	(* Switch S27 *)
	nAX5203DigitalInputs.3;
	

(* Axis 1-4 aktiv *)
	bLedH16 := ((Axis1.fbAxis.bMoveAbsBusy
					OR Axis2.fbAxis.bMoveAbsBusy
						OR Axis3.fbAxis.bMoveAbsBusy
							OR Axis4.fbAxis.bMoveAbsBusy)
				AND bClock500ms)
				OR (Axis1.fbAxis.bMoveAbsDone
					AND Axis2.fbAxis.bMoveAbsDone
						AND Axis3.fbAxis.bMoveAbsDone
							AND Axis4.fbAxis.bMoveAbsDone);

(* Axis 1-4 coupled *)
	bLedH17 := ((stAxis1.Status.Coupled
					OR stAxis2.Status.Coupled
						OR stAxis3.Status.Coupled
							OR stAxis4.Status.Coupled)
				AND bClock500ms)
				OR bSwitchS17;
				
(* Axis 1-4 reversing sequence busy *)		
	bLedH20 := (Axis1.fbAxis.bRevSeqBusy
					OR Axis2.fbAxis.bRevSeqBusy
						OR Axis3.fbAxis.bRevSeqBusy
							OR Axis4.fbAxis.bRevSeqBusy)
				AND bClock500ms;

(* Axis 1-4 error detectet *)
	bLedH21 := (stAxis1.Status.Error
					OR stAxis2.Status.Error
						OR stAxis3.Status.Error
							OR stAxis4.Status.Error)
				AND bClock500ms;

(* End *)

END_PROGRAM

// ---- POUs/Motion/Axis1.TcPOU
PROGRAM Axis1
VAR

	sAxisDescription						:STRING	:= 'Axis 1 - EL7037 - AS1020-0120';	

(* Axis - basic functions *)
	fbAxis									:FB_Axis;
	fMoveAbsPosition						:LREAL;				(* Target position *)
	fMoveAbsVelocity						:LREAL	:= 500.0;	(* Target speed axis 1 max. 3600.0 Degree/s *)
	bStartMoveAbs							:BOOL;
	bMoveAbsBusy							:BOOL;
	bMoveAbsDone							:BOOL;
	bAxisErr								:BOOL;
	nAxisErrId								:DWORD;
	bReset									:BOOL;
	bStop									:BOOL;
	bStopAxisDone							:BOOL;
	bStopAxisBusy							:BOOL;
	bRevSeqStart							:BOOL;
	bStartparameterSet						:BOOL;
	
(* Test - change target position *)
	bTestChangeTargetPos					:BOOL;				(* Test - change target position *)
	bMaxPositionReached						:BOOL;
	
(* Homing *)
	fbHomingAxis							:MC_Home;
	fHomingPosition							:LREAL	:= 331.00;

(* Touch Probe *)
	fbTouchProbe							:MC_TouchProbe;
	stTriggerInput							:TRIGGER_REF;
	bTouchProbeDone							:BOOL;
	bTouchProbeBusy							:BOOL;
	bTouchProbeComAb						:BOOL;
	bTouchProbeErr							:BOOL;
	bTouchProbeErrId						:UDINT;
	fRecordedPosition 						:LREAL;
	stRecordedData							:MC_TouchProbeRecordedData;	

(* Couple Axis on Handwheel *)
	fbGearIn								:MC_GearIn;
	bGearInDone								:BOOL;
	bAxisCoupled							:BOOL;

(* Uncouple Axis *)
	fbGearOut								:MC_GearOut;
	bGearOutDone							:BOOL;

END_VAR
(* End *)

(* Axis 1 *)

(* Axis - basic functions  *)

	IF NOT bStartparameterSet
	THEN
		(* Startup Parameter reversing sequence *)
		fbAxis.fRevSeqTargetPos1	:= 720.0;
		fbAxis.fRevSeqTargetVelo1	:= 500.0;
		fbAxis.fRevSeqTargetPos2	:= 0.0;
		fbAxis.fRevSeqTargetVelo2	:= 3000.0;
		fbAxis.nRevSeqIdleTime		:= 500;
		bStartparameterSet			:= TRUE;
	END_IF
		
	fbAxis(
		bPowerEnable		:= 	bSwitchS12,
		fPowerOverride		:= 	F_Scaling(nAnalogInR10, 100.0, 32767.0),
		bMoveAbsExecute		:= 	(bStartMoveAbs OR bSwitchS16) AND NOT stAxis1.Status.Coupled,
		fMoveAbsPosition	:= 	fMoveAbsPosition,
		fMoveAbsVelocity	:= 	fMoveAbsVelocity,
		bReset				:= 	bReset OR bSwitchS21,
		bStopAxis			:= 	bStop,
		bRevSeqStart		:=  (bSwitchS20 OR bRevSeqStart) AND fbAxis.bPowerStatus, 
		stAxis				:= 	stAxis1,
		bPowerStatus		=> 	bLedH12,
		bMoveAbsDone		=> 	bMoveAbsDone,
		bMoveAbsBusy		=> 	bMoveAbsBusy,
		bAxisErr			=> 	bAxisErr,
		nAxisErrId			=> 	nAxisErrId,
		bStopAxisDone		=> 	bStopAxisDone,
		bStopAxisBusy		=> 	bStopAxisBusy);
		

(* Test - change target position - Axis *)
	IF bTestChangeTargetPos
		AND (fMoveAbsPosition <= stAxis1.NcToPlc.ActPos)
			AND NOT bMaxPositionReached
	THEN
		fMoveAbsPosition := fMoveAbsPosition + 180.0;
	ELSE
		IF bTestChangeTargetPos
			AND (fMoveAbsPosition >= 3600.0)
		THEN
			fMoveAbsPosition 	:= 0.0;
			bMaxPositionReached	:= TRUE;
		END_IF
	END_IF

	IF bTestChangeTargetPos
		AND (stAxis1.NcToPlc.ActPos < 1.0)
	THEN
		bMaxPositionReached	:= FALSE;
	END_IF

	IF bSwitchS17
	THEN
		bMaxPositionReached	:= FALSE;
		fMoveAbsPosition 	:= 0.0;
	END_IF
	
(* Homing Axis *)
	fbHomingAxis(
		Execute			:= 	bSwitchS23 AND fbAxis.bPowerStatus,
		Position		:= 	fHomingPosition,
		HomingMode		:= 	MC_DefaultHoming,
		BufferMode		:= 	,
		Options			:= 	,
		bCalibrationCam	:= 	bStepperReferenceCam,
		Axis			:= 	stAxis1,
		Done			=> 	,
		Busy			=> 	,
		Active			=> 	,
		CommandAborted	=> 	,
		Error			=> 	,
		ErrorID			=> 	);
		
		
	bLedH23 :=	(bClock1s 
					AND NOT stAxis1.Status.Homed
					AND fbAxis.bPowerStatus
					AND NOT fbHomingAxis.Busy)
				OR (bClock500ms 
					AND fbHomingAxis.Busy)
				OR fbHomingAxis.Done;
					

(* Touch Probe *)
	stTriggerInput.EncoderID 		:= 1;
	stTriggerInput.TouchProbe 		:= TouchProbe1;
	stTriggerInput.SignalSource 	:= SignalSource_Default;
	stTriggerInput.Edge 			:= RisingEdge;
	stTriggerInput.Mode 			:= TOUCHPROBEMODE_SINGLE;
	stTriggerInput.ModuloPositions 	:= FALSE;

	fbTouchProbe(
		Execute			:= 	bSwitchS24,
		WindowOnly		:= 	,
		FirstPosition	:= 	,
		LastPosition	:= 	,
		Axis			:= 	stAxis1,
		TriggerInput	:= 	stTriggerInput,
		Done			=> 	bTouchProbeDone,
		Busy			=> 	bTouchProbeBusy,
		CommandAborted	=> 	bTouchProbeComAb,
		Error			=> 	bTouchProbeErr,
		ErrorID			=> 	bTouchProbeErrId,
		RecordedPosition=> 	fRecordedPosition,
		RecordedData	=>	stRecordedData);
	
	bLedH24 :=	(bClock500ms 
					AND fbTouchProbe.Busy)
						OR fbTouchProbe.Done;

(* Couple Axis on Handwheel *)
	fbGearIn(
		Execute			:= 	bHandwheelSwitchS28,
		RatioNumerator	:= 	1,
		RatioDenominator:= 	1,
		Acceleration	:= 	,
		Deceleration	:= 	,
		Jerk			:= 	,
		BufferMode		:= 	,
		Options			:= 	,
		Master			:= 	stAxis5,
		Slave			:= 	stAxis1,
		InGear			=> 	bGearInDone,
		Busy			=> 	,
		Active			=> 	,
		CommandAborted	=> 	,
		Error			=> 	,
		ErrorID			=> 	);

(* Axis coupled *)
	bAxisCoupled := stAxis1.Status.Coupled;

(* Uncouple Axis *)
	fbGearOut(
		Execute	:= 	bSwitchS17,
		Options	:= 	,
		Slave	:= 	stAxis1,
		Done	=> 	bGearOutDone,
		Busy	=> 	,
		Error	=> 	,
		ErrorID	=> 	);
	
(* End *)

END_PROGRAM

// ---- POUs/Motion/Components/FB_Axis.TcPOU
FUNCTION_BLOCK FB_Axis
VAR_INPUT
	
	bPowerEnable							:BOOL;
	fPowerOverride							:LREAL;
	bMoveAbsExecute							:BOOL;
	fMoveAbsPosition						:LREAL;
	fMoveAbsVelocity						:LREAL;
	bReset									:BOOL;
	bStopAxis								:BOOL;
	bRevSeqStart							:BOOL;
	bRevSeqStop								:BOOL;
	fRevSeqTargetPos1						:LREAL; 
	fRevSeqTargetVelo1						:LREAL;	 
	fRevSeqTargetPos2						:LREAL;	 
	fRevSeqTargetVelo2						:LREAL; 
	nRevSeqIdleTime							:UINT;
	
END_VAR
VAR_OUTPUT

	bPowerStatus							:BOOL;
	bMoveAbsDone							:BOOL;
	bMoveAbsBusy							:BOOL;
	bAxisErr								:BOOL;
	nAxisErrId								:DWORD;
	bStopAxisDone							:BOOL;
	bStopAxisBusy							:BOOL;
	bRevSeqDone								:BOOL;
	bRevSeqBusy								:BOOL;
	
END_VAR
VAR_IN_OUT

	stAxis									:Axis_Ref;

END_VAR
VAR

	fbMcPower								:MC_Power;
	fbMoveAbsolute							:MC_MoveAbsolute;
	fbReadAxisError							:MC_ReadAxisError;
	fbReset									:MC_Reset;
	fbStop									:MC_Stop;
	fbReversingSequence						:FB_ReversingSequence;

END_VAR
(* End *)

(* FB_Axis *)

(* Read status of the axis *)
	stAxis.ReadStatus();

(* Enable axis *)
	fbMcPower(
		Enable			:= 	bPowerEnable,
		Enable_Positive	:= 	bPowerEnable,
		Enable_Negative	:= 	bPowerEnable,
		Override		:= 	fPowerOverride,
		Axis			:= 	stAxis,
		Status			=> 	bPowerStatus);

(* Start axis at an absolute position *)
	fbMoveAbsolute(
		Execute		:=	bMoveAbsExecute,
		Position	:=	fMoveAbsPosition,
		Velocity	:=	fMoveAbsVelocity,
		Axis		:=	stAxis,
		Done		=>	bMoveAbsDone,
		Busy		=>	bMoveAbsBusy);

(* Read the error code of the axis *)
	fbReadAxisError(
		Enable		:=	TRUE,
		Axis		:=	stAxis,
		AxisErrorID	=>	nAxisErrId);
		
	bAxisErr := nAxisErrId <> 0;

(* Reset axis in case of failure *)
	fbReset(
		Execute		:= 	bReset,
		Axis		:= 	stAxis);

(* Stop axis *)
	fbStop(
		Execute 	:=	bStopAxis,
		Axis		:=	stAxis,
		Done		=>	bStopAxisDone,
		Busy		=>	bStopAxisBusy);

(* Axis reversing sequence *)	
	fbReversingSequence(
		bStart				:= 	bRevSeqStart,
		bStop				:= 	bRevSeqStop,
		fTargetPosition1	:= 	fRevSeqTargetPos1,
		fTargetVelocity1	:= 	fRevSeqTargetVelo1,
		fTargetPosition2	:= 	fRevSeqTargetPos2,
		fTargetVelocity2	:= 	fRevSeqTargetVelo2,
		tIdleTime			:= 	TO_TIME(nRevSeqIdleTime),
		bDone				=> 	bRevSeqDone,
		bBusy				=> 	bRevSeqBusy,
		bErr				=> 	,
		nErrID				=> 	,
		stAxis				:= 	stAxis);
		
(* End *)

END_FUNCTION_BLOCK

// ---- POUs/Motion/Components/FB_ReversingSequence.TcPOU
FUNCTION_BLOCK FB_ReversingSequence
VAR_INPUT
	
	bStart									:BOOL;
	bStop									:BOOL;	
	fTargetPosition1						:LREAL;
	fTargetVelocity1						:LREAL;
	fTargetPosition2						:LREAL;
	fTargetVelocity2						:LREAL;
	tIdleTime								:TIME;
	
END_VAR
VAR_OUTPUT
	
	bDone									:BOOL;
	bBusy									:BOOL;
	bErr									:BOOL;
	nErrID									:UDINT;
	
END_VAR
VAR_IN_OUT

	stAxis									:Axis_Ref;

END_VAR
VAR
	
	eStateRevSeq							:E_AxisReversingSequence;
	eRevSeqErrStep							:E_AxisReversingSequence := eAxisRevSeq_NoError;
	fbTimerIdleTime							:TON;
	fbMoveAbsolute							:MC_MoveAbsolute;
	fbStop									:MC_Stop;

END_VAR
(* End *)

(* Reversing sequence axis *)

	CASE eStateRevSeq OF

		eAxisRevSeq_Start			:	(* Wait for start *)
		
			bDone := FALSE;
			bBusy := FALSE;
			
			IF bStart
			THEN

				bBusy 		 := TRUE;
				eStateRevSeq := eAxisRevSeq_Init;
				
			END_IF		


		eAxisRevSeq_Init			:	(* Initialize *)
		
			fbMoveAbsolute(
				Axis	 := stAxis, 
				Execute	 := FALSE);
				
			fbTimerIdleTime(
				IN	 	 :=	FALSE);
			
			fbStop(
				Axis	 :=	stAxis,
				Execute	 :=	FALSE);
				
			eStateRevSeq := eAxisRevSeq_AxisStartPos1;


		eAxisRevSeq_AxisStartPos1	:	(* Start axis to position 1 *)
		
			fbMoveAbsolute(
				Axis		:= stAxis, 
				Execute		:= TRUE, 
				Position	:= fTargetPosition1, 
				Velocity	:= fTargetVelocity1, 
				ErrorID		=> nErrID);
			
		
			IF NOT fbMoveAbsolute.Busy
				AND NOT fbMoveAbsolute.Error
			THEN
			
				fbMoveAbsolute(
					Axis		:= stAxis, 
					Execute		:= FALSE);
				eStateRevSeq := eAxisRevSeq_IdleTime1;

			ELSIF bStop
			THEN

				fbMoveAbsolute(
					Axis	 := stAxis, 
					Execute	 := FALSE);
				eStateRevSeq := eAxisRevSeq_AxisStop;

			ELSIF NOT fbMoveAbsolute.Busy
					AND fbMoveAbsolute.Error
			THEN

				eRevSeqErrStep := eStateRevSeq;
				eStateRevSeq   := eAxisRevSeq_ErrorStep;

			END_IF


		eAxisRevSeq_IdleTime1		:	(* delayed restart *)
		
			fbTimerIdleTime(
				IN	:=	TRUE, 
				PT	:= 	tIdleTime);

			IF NOT bStop			
				AND fbTimerIdleTime.Q 
			THEN

				fbTimerIdleTime(IN	:=	FALSE);
				eStateRevSeq := eAxisRevSeq_AxisStartPos2;

			ELSIF bStop
			THEN

				eStateRevSeq := eAxisRevSeq_Done;

			END_IF


		eAxisRevSeq_AxisStartPos2	:	(* Start axis to position 2 *)
		
			fbMoveAbsolute(
				Axis		:= stAxis, 
				Execute		:= TRUE, 
				Position	:= fTargetPosition2, 
				Velocity	:= fTargetVelocity2, 
				ErrorID		=> nErrID);
			
		
			IF NOT fbMoveAbsolute.Busy
				AND NOT fbMoveAbsolute.Error
			THEN
				fbMoveAbsolute(
					Axis	 := stAxis, 
					Execute	 := FALSE);
				eStateRevSeq := eAxisRevSeq_IdleTime2;

			ELSIF bStop
			THEN

				fbMoveAbsolute(
					Axis		:= stAxis, 
					Execute	:= FALSE);
				eStateRevSeq := eAxisRevSeq_AxisStop;

			ELSIF NOT fbMoveAbsolute.Busy
					AND fbMoveAbsolute.Error
			THEN

				eRevSeqErrStep := eStateRevSeq;
				eStateRevSeq   := eAxisRevSeq_ErrorStep;

			END_IF		


		eAxisRevSeq_IdleTime2		:	(* delayed restart*)

			fbTimerIdleTime(
				IN	:=	TRUE, 
				PT	:= 	tIdleTime);
				
			IF NOT bStop			
				AND fbTimerIdleTime.Q 
			THEN

				fbTimerIdleTime(IN	:=	FALSE);
				eStateRevSeq := eAxisRevSeq_Done;
				
			ELSIF bStop
			THEN
			
				eStateRevSeq := eAxisRevSeq_Done;
				
			END_IF
			
			
		eAxisRevSeq_AxisStop		:	(* Stop axis *)

			fbStop(
				Axis	:=	stAxis, 
				Execute	:=	TRUE, 
				ErrorID	=>	nErrID );
				
			IF (fbStop.Done
				OR fbStop.CommandAborted)
				AND NOT fbStop.Error
			THEN
				fbStop(
					Axis	:=	stAxis, 
					Execute	:=	FALSE);
				eStateRevSeq := eAxisRevSeq_Done;

			ELSIF NOT fbStop.Busy
					AND fbStop.Error
			THEN

				eRevSeqErrStep := eStateRevSeq;
				eStateRevSeq   := eAxisRevSeq_ErrorStep;

			END_IF			
				
			
		eAxisRevSeq_Done			:	(* Sequence done *)

			bDone := TRUE;
			
			IF NOT bStart
				AND NOT bStop
			THEN
				bDone 		 := FALSE;
				bBusy 		 := FALSE;
				eStateRevSeq := eAxisRevSeq_Start;
				
			ELSIF bStart
				AND NOT bStop
			THEN
				bDone 		 := FALSE;
				eStateRevSeq := eAxisRevSeq_AxisStartPos1;
			END_IF

			
		eAxisRevSeq_ErrorStep		:	(* Error step *)
		
			bErr := TRUE;
			nErrID;
			
			IF NOT bStart
				AND NOT bStop
			THEN
				bErr 		   := FALSE;
				nErrID		   := 0;
				eRevSeqErrStep := eAxisRevSeq_NoError;
				eStateRevSeq   := eAxisRevSeq_Start;
			END_IF

	ELSE

		(* If not a valid step is active, then put on start *)
		eRevSeqErrStep := eAxisRevSeq_NoError;
		eStateRevSeq   := eAxisRevSeq_Start;

	END_CASE

(* End *)

END_FUNCTION_BLOCK

// ---- POUs/Motion/Axis2.TcPOU
PROGRAM Axis2
VAR
	
	sAxisDescription						:STRING	:= 'Axis 2 - EL7201 - AM8111-0F20';	

(* Axis - basic functions *)
	fbAxis									:FB_Axis;
	fMoveAbsPosition						:LREAL;				(* Target position *)
	fMoveAbsVelocity						:LREAL	:= 500.0;	(* Target speed axis 2 max. 10000.0 Degree/s *)
	bStartMoveAbs							:BOOL;
	bMoveAbsBusy							:BOOL;
	bMoveAbsDone							:BOOL;
	bAxisErr								:BOOL;
	nAxisErrId								:DWORD;
	bReset									:BOOL;
	bStop									:BOOL;
	bStopAxisDone							:BOOL;
	bStopAxisBusy							:BOOL;
	bRevSeqStart							:BOOL;
	bStartparameterSet						:BOOL;
	
(* Test - change target position - Axis *)
	bTestChangeTargetPos					:BOOL;				(* Test - change target position *)
	bMaxPositionReached						:BOOL;

(* Couple Axis on Handwheel) *)
	fbGearIn								:MC_GearIn;
	bGearInDone								:BOOL;
	bAxisCoupled							:BOOL;

(* Uncouple Axis *)
	fbGearOut								:MC_GearOut;
	bGearOutDone							:BOOL;

END_VAR
(* End *)

(* Axis 2 *)

(* Axis - basic functions  *)

	IF NOT bStartparameterSet
	THEN
		(* Startup Parameter reversing sequence *)
		fbAxis.fRevSeqTargetPos1	:= 1800.0;
		fbAxis.fRevSeqTargetVelo1	:= 1500.0;
		fbAxis.fRevSeqTargetPos2	:= 0.0;
		fbAxis.fRevSeqTargetVelo2	:= 200.0;
		fbAxis.nRevSeqIdleTime		:= 500;
		bStartparameterSet			:=TRUE;
	END_IF
		
	fbAxis(
		bPowerEnable		:= 	bSwitchS13,
		fPowerOverride		:= 	F_Scaling(nAnalogInR10, 100.0, 32767.0),
		bMoveAbsExecute		:= 	(bStartMoveAbs OR bSwitchS16) AND NOT stAxis2.Status.Coupled,
		fMoveAbsPosition	:= 	fMoveAbsPosition,
		fMoveAbsVelocity	:= 	fMoveAbsVelocity,
		bReset				:= 	bReset OR bSwitchS21,
		bStopAxis			:= 	bStop,
		bRevSeqStart		:=  (bSwitchS20 OR bRevSeqStart) AND fbAxis.bPowerStatus, 
		stAxis				:= 	stAxis2,
		bPowerStatus		=> 	bLedH13,
		bMoveAbsDone		=> 	bMoveAbsDone,
		bMoveAbsBusy		=> 	bMoveAbsBusy,
		bAxisErr			=> 	bAxisErr,
		nAxisErrId			=> 	nAxisErrId,
		bStopAxisDone		=> 	bStopAxisDone,
		bStopAxisBusy		=> 	bStopAxisBusy);

(* Test - change target position - Axis *)
	IF bTestChangeTargetPos
		AND (fMoveAbsPosition <= stAxis2.NcToPlc.ActPos)
			AND NOT bMaxPositionReached
	THEN
		fMoveAbsPosition := fMoveAbsPosition + 180.0;
	ELSE
		IF bTestChangeTargetPos
			AND (fMoveAbsPosition >= 3600.0)
		THEN
			fMoveAbsPosition 	:= 0.0;
			bMaxPositionReached	:= TRUE;
		END_IF
	END_IF

	IF bTestChangeTargetPos
		AND (stAxis2.NcToPlc.ActPos < 1.0)
	THEN
		bMaxPositionReached	:= FALSE;
	END_IF

	IF bSwitchS17
	THEN
		bMaxPositionReached	:= FALSE;
		fMoveAbsPosition 	:= 0.0;
	END_IF
	
(* Couple Axis on Handwheel *)
	fbGearIn(
		Execute			:= 	bHandwheelSwitchS28,
		RatioNumerator	:= 	1,
		RatioDenominator:= 	1,
		Acceleration	:= 	,
		Deceleration	:= 	,
		Jerk			:= 	,
		BufferMode		:= 	,
		Options			:= 	,
		Master			:= 	stAxis5,
		Slave			:= 	stAxis2,
		InGear			=> 	bGearInDone,
		Busy			=> 	,
		Active			=> 	,
		CommandAborted	=> 	,
		Error			=> 	,
		ErrorID			=> 	);

(* Axis coupled *)
	bAxisCoupled := stAxis2.Status.Coupled;

(* Uncouple Axis *)
	fbGearOut(
		Execute	:= 	bSwitchS17,
		Options	:= 	,
		Slave	:= 	stAxis2,
		Done	=> 	bGearOutDone,
		Busy	=> 	,
		Error	=> 	,
		ErrorID	=> 	);
	
(* End *)

END_PROGRAM

// ---- POUs/Motion/Axis3.TcPOU
PROGRAM Axis3
VAR
	
	sAxisDescription						:STRING	:= 'Axis 3 - AX5203-A - AM8111-0F10';	

(* Axis - basic functions *)
	fbAxis									:FB_AxisAX5xxx;
	fMoveAbsPosition						:LREAL;				(* Target position *)
	fMoveAbsVelocity						:LREAL	:= 500.0;	(* Target speed axis 3 max. 18000.0 Degree/s *)
	bStartMoveAbs							:BOOL;
	bMoveAbsBusy							:BOOL;
	bMoveAbsDone							:BOOL;
	bAxisErr								:BOOL;
	nAxisErrId								:DWORD;
	bReset									:BOOL;
	bStop									:BOOL;
	bStopAxisDone							:BOOL;
	bStopAxisBusy							:BOOL;
	bRevSeqStart							:BOOL;
	bStartparameterSet						:BOOL;
	
(* Test - change target position - Axis 3 *)
	bTestChangeTargetPos					:BOOL;				(* Test - change target position *)
	bMaxPositionReached						:BOOL;	

(* Couple Axis 3 on Axis 5 (Handwheel) *)
	fbGearIn								:MC_GearIn;
	bGearInDone								:BOOL;
	bAxisCoupled							:BOOL;

(* Uncouple Axis 3 *)
	fbGearOut								:MC_GearOut;
	bGearOutDone							:BOOL;
	
(*Superimposed and Buffered Moves*)
	mv_Axis3Abs : MC_MoveAbsolute;
	mv_Axis3Rel : MC_MoveRelative;
	iMstrMvMode2	: INT;
	bMvMstr2		: BOOL;
	lrMstrTarg2		: LREAL := 90;
	lrMstrVelo2		: LREAL := 10;
	mv_MasterSprImp	: MC_MoveSuperImposed;
	bMvMstr3		: BOOL;
	lrMstrTarg3		: LREAL := 90;

END_VAR
(* End *)

(* Axis 3 *)

(* Axis - basic functions  *)

	IF NOT bStartparameterSet
	THEN
		(* Startup Parameter reversing sequence *)
		fbAxis.fRevSeqTargetPos1	:= 720.0;
		fbAxis.fRevSeqTargetVelo1	:= 5000.0;
		fbAxis.fRevSeqTargetPos2	:= 0.0;
		fbAxis.fRevSeqTargetVelo2	:= 5000.0;
		fbAxis.nRevSeqIdleTime		:= 250;
		bStartparameterSet			:=TRUE;
	END_IF
		
	fbAxis(
		bPowerEnable		:= 	bSwitchS14,
		fPowerOverride		:= 	F_Scaling(aOsAnalogInR11[0], 100.0, 32767.0),
		bMoveAbsExecute		:= 	(bStartMoveAbs OR bSwitchS16) AND NOT stAxis3.Status.Coupled,
		fMoveAbsPosition	:= 	fMoveAbsPosition,
		fMoveAbsVelocity	:= 	fMoveAbsVelocity,
		bReset				:= 	bReset OR bSwitchS21,
		bStopAxis			:= 	bStop,
		bRevSeqStart		:=  (bSwitchS20 OR bRevSeqStart) AND fbAxis.bPowerStatus, 
		stAxis				:= 	stAxis3,
		bPowerStatus		=> 	bLedH14,
		bMoveAbsDone		=> 	bMoveAbsDone,
		bMoveAbsBusy		=> 	bMoveAbsBusy,
		bAxisErr			=> 	bAxisErr,
		nAxisErrId			=> 	nAxisErrId,
		bStopAxisDone		=> 	bStopAxisDone,
		bStopAxisBusy		=> 	bStopAxisBusy);

(* Test - change target position - Axis *)
	IF bTestChangeTargetPos
		AND (fMoveAbsPosition <= stAxis3.NcToPlc.ActPos)
			AND NOT bMaxPositionReached
	THEN
		fMoveAbsPosition := fMoveAbsPosition + 180.0;
	ELSE
		IF bTestChangeTargetPos
			AND (fMoveAbsPosition >= 3600.0)
		THEN
			fMoveAbsPosition 	:= 0.0;
			bMaxPositionReached	:= TRUE;
		END_IF
	END_IF

	IF bTestChangeTargetPos
		AND (stAxis3.NcToPlc.ActPos < 1.0)
	THEN
		bMaxPositionReached	:= FALSE;
	END_IF

	IF bSwitchS17
	THEN
		bMaxPositionReached	:= FALSE;
		fMoveAbsPosition 	:= 0.0;
	END_IF
	
(* Couple Axis on Handwheel *)
	fbGearIn(
		Execute			:= 	bHandwheelSwitchS28,
		RatioNumerator	:= 	1,
		RatioDenominator:= 	1,
		Acceleration	:= 	,
		Deceleration	:= 	,
		Jerk			:= 	,
		BufferMode		:= 	,
		Options			:= 	,
		Master			:= 	stAxis5,
		Slave			:= 	stAxis3,
		InGear			=> 	bGearInDone,
		Busy			=> 	,
		Active			=> 	,
		CommandAborted	=> 	,
		Error			=> 	,
		ErrorID			=> 	);

(* Axis coupled *)
	bAxisCoupled := stAxis3.Status.Coupled;

(* Uncouple Axis *)
	fbGearOut(
		Execute	:= 	bSwitchS17,
		Options	:= 	,
		Slave	:= 	stAxis3,
		Done	=> 	bGearOutDone,
		Busy	=> 	,
		Error	=> 	,
		ErrorID	=> 	);

		
(*Buffered Move*)
	mv_Axis3Abs(
		Axis:= stAxis3, 
		Execute:= iMstrMvMode2=0 AND bMvMstr2, 
		Position:= lrMstrTarg2, 
		Velocity:= lrMstrVelo2);
		
	mv_Axis3Rel(	
		Axis:= stAxis3, 
		Execute:= iMstrMvMode2=1 AND bMvMstr2, 
		Distance:= lrMstrTarg2, 
		Velocity:= lrMstrVelo2);
		
IF (NOT(mv_Axis3Abs.Busy) AND NOT(mv_Axis3Rel.busy)) THEN
	bMvMstr2:=FALSE;
END_IF

(*Superimposed Move*)
mv_MasterSprImp(
	Axis:= stAxis3, 
	Execute:= bMvMstr3, 
	Mode:= SUPERPOSITIONMODE_VELOREDUCTION_ADDITIVEMOTION, 
	Distance:= lrMstrTarg3, 
	// assume max velo is 2000 (config parameter)
	VelocityDiff:= 2000-stAxis3.NcToPlc.SetVelo, 
	Acceleration:= , 
	Deceleration:= , 
	Jerk:= , 
	VelocityProcess:= stAxis3.NcToPlc.SetVelo, 
	// use 75% of remaining distance to 'catch up'
	Length:= (stAxis3.NcToPlc.TargetPos-stAxis3.NcToPlc.ActPos)*0.75);
			
(* End *)

END_PROGRAM

// ---- POUs/Motion/Components/FB_AxisAX5xxx.TcPOU
FUNCTION_BLOCK FB_AxisAX5xxx
VAR_INPUT

	bPowerEnable							:BOOL;
	fPowerOverride							:LREAL;
	bMoveAbsExecute							:BOOL;
	fMoveAbsPosition						:LREAL;
	fMoveAbsVelocity						:LREAL;
	bReset									:BOOL;
	bStopAxis								:BOOL;
	bRevSeqStart							:BOOL;
	bRevSeqStop								:BOOL;
	fRevSeqTargetPos1						:LREAL; 
	fRevSeqTargetVelo1						:LREAL;	 
	fRevSeqTargetPos2						:LREAL;	 
	fRevSeqTargetVelo2						:LREAL; 
	nRevSeqIdleTime							:UINT;
	
END_VAR
VAR_OUTPUT

	bPowerStatus							:BOOL;
	bMoveAbsDone							:BOOL;
	bMoveAbsBusy							:BOOL;
	bAxisErr								:BOOL;
	nAxisErrId								:DWORD;
	bStopAxisDone							:BOOL;
	bStopAxisBusy							:BOOL;
	bRevSeqDone								:BOOL;
	bRevSeqBusy								:BOOL;
	
END_VAR
VAR_IN_OUT

	stAxis									:Axis_Ref;

END_VAR
VAR

	fbMcPower								:MC_Power;
	fbMoveAbsolute							:MC_MoveAbsolute;
	fbReadAxisError							:MC_ReadAxisError;
	fbReset									:MC_Reset_Ax5xxx;
	fbStop									:MC_Stop;
	fbReversingSequence						:FB_ReversingSequence;

END_VAR
(* End *)

(* FB_Axis AX5xxx *)

(* Read status of the axis *)
	stAxis.ReadStatus();

(* Enable axis *)
	fbMcPower(
		Enable			:= 	bPowerEnable,
		Enable_Positive	:= 	bPowerEnable,
		Enable_Negative	:= 	bPowerEnable,
		Override		:= 	fPowerOverride,
		Axis			:= 	stAxis,
		Status			=> 	bPowerStatus);

(* Start axis at an absolute position *)
	fbMoveAbsolute(
		Execute		:=	bMoveAbsExecute,
		Position	:=	fMoveAbsPosition,
		Velocity	:=	fMoveAbsVelocity,
		Axis		:=	stAxis,
		Done		=>	bMoveAbsDone,
		Busy		=>	bMoveAbsBusy);

(* Read the error code of the axis *)
	fbReadAxisError(
		Enable		:=	TRUE,
		Axis		:=	stAxis,
		AxisErrorID	=>	nAxisErrId);

	bAxisErr := nAxisErrId <> 0;

(* Reset axis in case of failure *)
	fbReset(
		Execute		:= 	bReset,
		Axis		:= 	stAxis);

(* Stop axis *)
	fbStop(
		Execute 	:=	bStopAxis,
		Axis		:=	stAxis,
		Done		=>	bStopAxisDone,
		Busy		=>	bStopAxisBusy);

(* Axis reversing sequence *)	
	fbReversingSequence(
		bStart				:= 	bRevSeqStart,
		bStop				:= 	bRevSeqStop,
		fTargetPosition1	:= 	fRevSeqTargetPos1,
		fTargetVelocity1	:= 	fRevSeqTargetVelo1,
		fTargetPosition2	:= 	fRevSeqTargetPos2,
		fTargetVelocity2	:= 	fRevSeqTargetVelo2,
		tIdleTime			:= 	TO_TIME(nRevSeqIdleTime),
		bDone				=> 	bRevSeqDone,
		bBusy				=> 	bRevSeqBusy,
		bErr				=> 	,
		nErrID				=> 	,
		stAxis				:= 	stAxis);
		
(* End *)

END_FUNCTION_BLOCK

// ---- POUs/Motion/Components/MC_Reset_Ax5xxx.TcPOU
FUNCTION_BLOCK MC_Reset_Ax5xxx
VAR_INPUT

	Execute									:BOOL;

END_VAR
VAR_IN_OUT

	Axis	 								:AXIS_REF;

END_VAR
VAR_OUTPUT

	Done									:BOOL;
	Busy									:BOOL;
	Error									:BOOL;
	ErrorId									:DWORD;

END_VAR
VAR

	bDriveProtected							:BOOL;
	bDriveDeviceError						:BOOL;
	bDriveIoDataInvalid						:BOOL;
	bDriveError								:BOOL;

	fbNcReset								:MC_Reset;
	fbSoEReset								:FB_SoEReset;

	eStateResetSeq							:E_McResetStatus;
	eResetSeqErrStep						:E_McResetStatus := eMcReset_NoError;

END_VAR
(* End *)

(* MC_Reset_Ax5xxx *)

(* Evaluate messages *)
	bDriveProtected 	:= TO_BOOL(Axis.NcToPlc.StateDWord.5);
	bDriveDeviceError   := TO_BOOL(Axis.NcToPlc.StateDWord.28);
	bDriveIoDataInvalid	:= TO_BOOL(Axis.NcToPlc.StateDWord.30);
	bDriveError			:= TO_BOOL(Axis.NcToPlc.StateDWord.31);

	
(* Reset sequence *)
	CASE eStateResetSeq OF
	
		eMcReset_Start			:	(* Wait for start *)
		
				Busy := FALSE;
				Done := FALSE;
	
				IF Execute
				THEN
				
					Busy := TRUE;
					eStateResetSeq := eMcReset_Init;

				END_IF


		eMcReset_Init			:	(* Initialize *)
			
				fbSoEReset(	
					NetId		:=	'',
					Execute		:=	FALSE,
					Timeout		:=	T#12S,
					Axis		:=	Axis);

				fbNcReset(	
					Execute		:=	FALSE,
					Axis		:=	Axis);

				eStateResetSeq 		:= eMcReset_ResetHardware;

	
		eMcReset_ResetHardware	:	(* Reset hardware *)
		
				fbSoEReset(	
					NetId	:=	'' ,
					Execute	:=	Execute
									AND (bDriveDeviceError
										OR bDriveIoDataInvalid),
					Timeout	:=	T#12S ,
					Axis	:=	Axis);
	
				IF NOT fbSoEReset.Busy
					AND NOT fbSoEReset.Error
				THEN
	
					fbSoEReset(	
						NetId	:=	'',
						Execute	:=	FALSE,
						Timeout	:=	T#12S,
						Axis	:=	Axis);
	
					eStateResetSeq := eMcReset_ResetNc;
	
				ELSIF NOT fbSoEReset.Busy
					AND fbSoEReset.Error
				THEN

					eResetSeqErrStep := eStateResetSeq;
					eStateResetSeq   := eMcReset_ErrorStep;
	
				END_IF


		eMcReset_ResetNc		:	(* Reset NC *)
		
				fbNcReset(	
					Execute	:=	Execute
									AND bDriveError
										AND NOT bDriveDeviceError
											AND NOT fbSoEReset.Busy
												AND NOT bDriveProtected,
					Axis	:=	Axis);
	
				IF NOT fbNcReset.Busy
					AND NOT fbNcReset.Error
				THEN
	
					fbNcReset(	
						Execute	:=	FALSE,
						Axis	:=	Axis);
	
					eStateResetSeq := eMcReset_Done;

				ELSIF NOT fbNcReset.Busy
					AND fbNcReset.Error
				THEN

					eResetSeqErrStep := eStateResetSeq;
					eStateResetSeq   := eMcReset_ErrorStep;
	
				END_IF
				
	
		eMcReset_Done			:	(* Reset done *)
		
				Busy := FALSE;
				Done := TRUE;
	
				IF NOT Execute
				THEN
					eStateResetSeq := eMcReset_Start;
				END_IF


		eMcReset_ErrorStep			:	(* Error step *)

			IF NOT Execute
			THEN
				eResetSeqErrStep := eMcReset_NoError;
				eStateResetSeq   := eMcReset_Start;
			END_IF


	ELSE

		(* If not a valid step is active, then put on start *)
		eResetSeqErrStep := eMcReset_NoError;
		eStateResetSeq 	 := eMcReset_Start;

	END_CASE

	Error	:= bDriveError
					OR bDriveDeviceError;

	ErrorId	:= Axis.NcToPlc.ErrorCode;

(* End *)

END_FUNCTION_BLOCK

// ---- POUs/Motion/Axis4.TcPOU
PROGRAM Axis4
VAR
	
	sAxisDescription						:STRING	:= 'Axis 4 - AX5203-B - AM8111-0F21';	

(* Axis - basic functions *)
	fbAxis									:FB_AxisAX5xxx;
	fMoveAbsPosition						:LREAL;				(* Target position *)
	fMoveAbsVelocity						:LREAL	:= 500.0;	(* Target speed axis 3 max. 18000.0 Degree/s *)
	bStartMoveAbs							:BOOL;
	bMoveAbsBusy							:BOOL;
	bMoveAbsDone							:BOOL;
	bAxisErr								:BOOL;
	nAxisErrId								:DWORD;
	bReset									:BOOL;
	bStop									:BOOL;
	bStopAxisDone							:BOOL;
	bStopAxisBusy							:BOOL;
	bRevSeqStart							:BOOL;
	bStartparameterSet						:BOOL;
	
(* Test - change target position - Axis 4 *)
	bTestChangeTargetPos					:BOOL;				(* Test - change target position *)
	bMaxPositionReached						:BOOL;
		
(* Couple Axis 4 on Axis 5 (Handwheel) *)
	fbGearIn								:MC_GearIn;
	bGearInDone								:BOOL;
	bAxisCoupled							:BOOL;

(* Uncouple Axis 4 *)
	fbGearOut								:MC_GearOut;
	bGearOutDone							:BOOL;
	
END_VAR
(* End *)

(* Axis 4 *)

(* Axis - basic functions  *)	

	IF NOT bStartparameterSet
	THEN
		(* Startup Parameter reversing sequence *)
		fbAxis.fRevSeqTargetPos1	:= 7200.0;
		fbAxis.fRevSeqTargetVelo1	:= 9000.0;
		fbAxis.fRevSeqTargetPos2	:= 0.0;
		fbAxis.fRevSeqTargetVelo2	:= 5000.0;
		fbAxis.nRevSeqIdleTime		:= 600;
		bStartparameterSet			:=TRUE;
	END_IF
		
	fbAxis(
		bPowerEnable		:= 	bSwitchS15,
		fPowerOverride		:= 	F_Scaling(aOsAnalogInR11[0], 100.0, 32767.0),
		bMoveAbsExecute		:= 	(bStartMoveAbs OR bSwitchS16) AND NOT stAxis4.Status.Coupled,
		fMoveAbsPosition	:= 	fMoveAbsPosition,
		fMoveAbsVelocity	:= 	fMoveAbsVelocity,
		bReset				:= 	bReset OR bSwitchS21,
		bStopAxis			:= 	bStop,
		bRevSeqStart		:=  (bSwitchS20 OR bRevSeqStart) AND fbAxis.bPowerStatus, 
		stAxis				:= 	stAxis4,
		bPowerStatus		=> 	bLedH15,
		bMoveAbsDone		=> 	bMoveAbsDone,
		bMoveAbsBusy		=> 	bMoveAbsBusy,
		bAxisErr			=> 	bAxisErr,
		nAxisErrId			=> 	nAxisErrId,
		bStopAxisDone		=> 	bStopAxisDone,
		bStopAxisBusy		=> 	bStopAxisBusy);

(* Test - change target position - Axis *)
	IF bTestChangeTargetPos
		AND (fMoveAbsPosition <= stAxis4.NcToPlc.ActPos)
			AND NOT bMaxPositionReached
	THEN
		fMoveAbsPosition := fMoveAbsPosition + 180.0;
	ELSE
		IF bTestChangeTargetPos
			AND (fMoveAbsPosition >= 3600.0)
		THEN
			fMoveAbsPosition 	:= 0.0;
			bMaxPositionReached	:= TRUE;
		END_IF
	END_IF

	IF bTestChangeTargetPos
		AND (stAxis4.NcToPlc.ActPos < 1.0)
	THEN
		bMaxPositionReached	:= FALSE;
	END_IF

	IF bSwitchS17
	THEN
		bMaxPositionReached	:= FALSE;
		fMoveAbsPosition	:= 0.0;
	END_IF
	
(* Couple Axis on Handwheel *)
	fbGearIn(
		Execute			:= 	bHandwheelSwitchS28,
		RatioNumerator	:= 	1,
		RatioDenominator:= 	1,
		Acceleration	:= 	,
		Deceleration	:= 	,
		Jerk			:= 	,
		BufferMode		:= 	,
		Options			:= 	,
		Master			:= 	stAxis5,
		Slave			:= 	stAxis4,
		InGear			=> 	bGearInDone,
		Busy			=> 	,
		Active			=> 	,
		CommandAborted	=> 	,
		Error			=> 	,
		ErrorID			=> 	);

(* Axis coupled *)
	bAxisCoupled := stAxis4.Status.Coupled;

(* Uncouple Axis *)
	fbGearOut(
		Execute	:= 	bSwitchS17,
		Options	:= 	,
		Slave	:= 	stAxis4,
		Done	=> 	bGearOutDone,
		Busy	=> 	,
		Error	=> 	,
		ErrorID	=> 	);
			
(* End *)

END_PROGRAM

// ---- POUs/EtherCatDiagnostic/DiagnosticEtherCAT.TcPOU
PROGRAM DiagnosticEtherCAT
VAR
END_VAR
(* End *)

(* Diagnosis of the EtherCat System *)

	fbDiagnosticEtherCAT(bEnable :=	TRUE);
	
(* End *)

END_PROGRAM

// ---- POUs/XFC/DcTimes.TcPOU
PROGRAM DcTimes
VAR
	(* Freeze reading *)
	bFreezeReading							:BOOL;

(* Actual distributed clock system times *)
	// F_GetActualDcTime
	dtActDcTime								:T_DCTIME64;
	stActDcTime								:DCTIMESTRUCT;
	sActDcTime								:STRING;

	// F_GetCurDcTaskTime
	dtActDcTaskTime							:T_DCTIME64;
	stActDcTaskTime							:DCTIMESTRUCT;
	sActDcTaskTime							:STRING;

END_VAR
(* End *)

(* Actual distributed clock system times *)

	IF NOT bFreezeReading
	THEN
		(* F_GetActualDcTime - This function supplies the current time*)
		dtActDcTime  	:= F_GetActualDcTime64();
		stActDcTime  	:= DCTIME64_TO_DCTIMESTRUCT(dtActDcTime);
		sActDcTime   	:= DCTIME64_TO_STRING(dtActDcTime);

		(* F_GetCurDcTaskTime - This function supplies the task target start time *)
		dtActDcTaskTime := F_GetCurDcTaskTime64();
		stActDcTaskTime := DCTIME64_TO_DCTIMESTRUCT(dtActDcTaskTime);
		sActDcTaskTime  := DCTIME64_TO_STRING(dtActDcTaskTime);
	END_IF

(* End *)

END_PROGRAM

// ---- POUs/XFC/AnalogOutputOversampling.TcPOU
PROGRAM AnalogOutputOversampling
VAR

(* Freeze writing *)
	bFreezeWriting							:BOOL; (* Force to freeze writing. You will be able to see actual oversampling output at the corresponding oversampling input termnal *)
	
(* EL4732 analog output Ch1 oversampling *)
	ni										:UINT;
	nCounter								:UINT;

(* Read task target start time *)
	dtActDcTime								:T_DCTIME;
	stActDcTime								:DCTIMESTRUCT;

END_VAR
(* End *)

(* EL4732 - analog output Ch1 oversampling - ongoing value 0 - 29900 *)


(* Read task target start time *)
	dtActDcTime := F_GetCurDcTaskTime();
	stActDcTime  := DCTIME_TO_DCTIMESTRUCT(dtActDcTime);


(* EL4732 analog output Ch1 oversampling *)
	IF NOT bFreezeWriting
	THEN 

		FOR ni := 0 TO 99 BY 1 DO
			IF nCounter >= 30000
			THEN
				nCounter := 0;
			END_IF
		
			aOsOutputToEL3702In2[ni] := UINT_TO_INT(nCounter);
			
			nCounter := nCounter + 100;
		END_FOR
	
	END_IF
		
(* End *)

END_PROGRAM

// ---- POUs/XFC/PositionCamTimeStampAxis2.TcPOU
PROGRAM PositionCamTimeStampAxis2
VAR
	
	(* Parameterize and control of the channel 1 *)
	stCamSwitchOptionsOut1					:ST_CamSwitchOptions;
	fbXfcPositionCamOut1					:XFC_PositionCam;
	stXfcPositionCamOut1					:OUTPUT_REF;
	stXfcPositionCamTrackRefOut1			:TRACK_REF;

	(* Parameterize and control of the channel 2 *)
	stCamSwitchOptionsOut2					:ST_CamSwitchOptions;
	fbXfcPositionCamOut2 					:XFC_PositionCam;
	stXfcPositionCamOut2					:OUTPUT_REF;
	stXfcPositionCamTrackRefOut2			:TRACK_REF;

	(* XFC_EL2252_V2 handles the output of a digital cam with the XFC time stamp terminal EL2252 *)	
	fbXfcEL2252								:XFC_EL2252_V2;
	
END_VAR
(* End *)

(* EL2252 - digital output Ch1 and Ch2 time stamp - position cam *)	

(* Ch1 - position cam axis 2  90 - 180 Degree
   Ch2 - position cam axis 2  30 - 90  Degree 
*)

(* Parameterize and control of the channel 1 *)
	stCamSwitchOptionsOut1.EncoderIndex		:= 0;	
	stCamSwitchOptionsOut1.UseAcceleration	:= FALSE;

	fbXfcPositionCamOut1(
		FirstOnPosition	:= 	90, 
		LastOnPosition	:= 	180, 
		Modulo			:= 	TRUE, 
		ModuloFactor	:= 	360.0, 
		OnCompensation	:= 	0.0, 
		OffCompensation	:= 	0.0, 
		Options			:= 	stCamSwitchOptionsOut1, 
		Error			=> 	, 
		ErrorID			=> 	, 
		Output			:= 	stXfcPositionCamOut1, 
		Axis			:= 	stAxis2);	

	stXfcPositionCamTrackRefOut1.ModuloPositions 	:= TRUE;
	stXfcPositionCamTrackRefOut1.ModuloFactor 		:= 360.0;
	stXfcPositionCamTrackRefOut1.OnCompensation 	:= 0.0;
	stXfcPositionCamTrackRefOut1.OffCompensation 	:= 0.0;
	stXfcPositionCamTrackRefOut1.Hysteresis 		:= 0.0;
	stXfcPositionCamTrackRefOut1.BreakRelease 		:= FALSE;
	stXfcPositionCamTrackRefOut1.Force 				:= FALSE;
	stXfcPositionCamTrackRefOut1.Disable 			:= FALSE;

	
(* Parameterize and control of the channel 2 *)
	stCamSwitchOptionsOut2.EncoderIndex		:= 0;	
	stCamSwitchOptionsOut2.UseAcceleration	:= FALSE;

	fbXfcPositionCamOut2(
		FirstOnPosition	:= 	30, 
		LastOnPosition	:= 	90, 
		Modulo			:= 	TRUE, 
		ModuloFactor	:= 	360.0, 
		OnCompensation	:= 	0.0, 
		OffCompensation	:= 	0.0, 
		Options			:= 	stCamSwitchOptionsOut2, 
		Error			=> 	, 
		ErrorID			=> 	, 
		Output			:= 	stXfcPositionCamOut2, 
		Axis			:= 	stAxis2);	

	stXfcPositionCamTrackRefOut2.ModuloPositions 	:= TRUE;
	stXfcPositionCamTrackRefOut2.ModuloFactor 		:= 360.0;
	stXfcPositionCamTrackRefOut2.OnCompensation 	:= 0.0;
	stXfcPositionCamTrackRefOut2.OffCompensation 	:= 0.0;
	stXfcPositionCamTrackRefOut2.Hysteresis 		:= 0.0;
	stXfcPositionCamTrackRefOut2.BreakRelease 		:= FALSE;
	stXfcPositionCamTrackRefOut2.Force 				:= FALSE;
	stXfcPositionCamTrackRefOut2.Disable 			:= FALSE;

	
(* XFC_EL2252_V2 handles the output of a digital cam with the XFC time stamp terminal EL2252 *)	
	fbXfcEL2252(
		ForceWhenLate		:= 	TRUE, 
		Error				=> 	, 
		ErrorID				=> 	, 
		ErrorOutputMissed	=> 	, 
		PrecisionReduced	=> 	, 
		Output1				:= 	stXfcPositionCamOut1, 
		Output2				:= 	stXfcPositionCamOut2, 
		TrackOptions1		:= 	stXfcPositionCamTrackRefOut1, 
		TrackOptions2		:= 	stXfcPositionCamTrackRefOut2, 
		EL2252				:= 	stEL2252);
	
(* End *)

END_PROGRAM

// ---- POUs/XFC/SignalLengthMeasurementCamAxis2.TcPOU
PROGRAM SignalLengthMeasurementCamAxis2
VAR
	
(* EL1262 digital input oversampling*)	
	aData									:ARRAY[0..9999] OF BOOL;	(* 0..9999 -> Maximum signal length 1000ms *)
	nDataArrayCounter						:UINT;

	ni1										:UINT;						(* Loop index 1 *)
	ni2										:INT;						(* Loop index 2 *)

	bSignalRisingEdgeDetected				:BOOL;
	bSignalFallingEdgeDetected				:BOOL;
	nSignalRisingEdge						:UINT;
	nSignalFallingEdge						:UINT;

	fCurrentSpeedAxis						:LREAL;

	nSignalLengthMicroSec					:UDINT;
	tSignalLength							:LTIME;
	fSignalLengthDegree						:LREAL;

END_VAR
(* End *)

(* EL1262 - digital input Ch1 oversampling - signal length measurement *)	

(* evaluate the rising and falling edge *) 
	FOR ni1 := 0 TO 9 BY 1 DO
		(* detected the rising edge *) 
			IF aAxis2RefCamOs[ni1] = TRUE
				AND NOT bSignalRisingEdgeDetected
			THEN
				bSignalRisingEdgeDetected  := TRUE;
				bSignalFallingEdgeDetected := FALSE;

				(* Save the storage agency of the rising edge *)
				nSignalRisingEdge 		   := ni1;
				
				(* Save the current speed of the axis *)
				fCurrentSpeedAxis 		   := stAxis2.NcToPlc.ActVelo;
				
				(* Reset the data array *)
				FOR ni2 := 0 TO 9999 BY 1 DO
					aData[ni2] := 0;
				END_FOR
	
				nDataArrayCounter := 0;
			END_IF
	
		(* detected the falling edge *) 
			IF aAxis2RefCamOs[ni1] = FALSE
				AND bSignalRisingEdgeDetected
			THEN
				bSignalRisingEdgeDetected  := FALSE;
				bSignalFallingEdgeDetected := TRUE;

				(* Save the storage agency of the falling edge *)
				nSignalFallingEdge 		   := nDataArrayCounter + ni1;
			END_IF
	END_FOR

(* Save and evaluate the data *)
	IF bSignalRisingEdgeDetected
		OR bSignalFallingEdgeDetected
	THEN
		(* Save the data *)
			FOR ni1 := 0 TO 9 BY 1 DO
				aData[nDataArrayCounter] := aAxis2RefCamOs[ni1];
				nDataArrayCounter 	     := nDataArrayCounter + 1;
				
				IF nDataArrayCounter > 9999
				THEN
					nDataArrayCounter		   := 0;
					bSignalRisingEdgeDetected  := FALSE;
					bSignalFallingEdgeDetected := FALSE;
				END_IF
			END_FOR

		(* Evaluate the data *)
			IF bSignalFallingEdgeDetected
			THEN
				bSignalFallingEdgeDetected := FALSE;
			
				(* Calculate signal length in time *)
				nSignalLengthMicroSec 	   := UINT_TO_UDINT((nSignalFallingEdge - nSignalRisingEdge)) * 100;
				tSignalLength 		       := UDINT_TO_LTIME(nSignalLengthMicroSec * 1000);
	
				(* Calculate signal length in degree *)
				fSignalLengthDegree        := (fCurrentSpeedAxis / 1000000) * nSignalLengthMicroSec;
			END_IF
	END_IF

(* End *)

END_PROGRAM

// ---- POUs/XFC/TouchProbeTimeStampCamAxis2.TcPOU
PROGRAM TouchProbeTimeStampCamAxis2
VAR
	
(* Touch Probe - EL1252 *)
	sTimeStampPos 							:STRING;
	sTimeStampNeg							:STRING;

	stXfcTriggerRef							:XFC_TRIGGER_REF;
	fbXfcTouchProbe							:XFC_TouchProbe;
	fPositionTouch							:LREAL;

END_VAR
(* End *)

(* EL1252 - digital input Ch1 time stamp - touch probe *)

(* Current timestamp times *)
	sTimeStampPos := DCTIME_TO_STRING(stEL1252Ch1.TimeStampPos);
	sTimeStampNeg := DCTIME_TO_STRING(stEL1252Ch1.TimeStampNeg);

(* Fill structure with values *)
	stXfcTriggerRef.Signal					:= stEL1252Ch1.Input;
	stXfcTriggerRef.TimestampRisingEdge 	:= stEL1252Ch1.TimeStampPos.dwLowPart;
	stXfcTriggerRef.TimestampFallingEdge 	:= stEL1252Ch1.TimeStampNeg.dwLowPart;
	stXfcTriggerRef.Edge					:= RisingEdge;								(* FallingEdge *)				
	stXfcTriggerRef.FreeRun					:= TRUE;
	stXfcTriggerRef.EncoderIndex			:= 0;
	stXfcTriggerRef.ModuloPositions			:= TRUE;
	stXfcTriggerRef.ModuloFactor			:= 360.0;

(* Evaluate the time stamp *)
	fbXfcTouchProbe(
		Axis				:= 	stAxis2,
		TriggerInput		:= 	stXfcTriggerRef,
		Execute				:= 	TRUE,
		WindowOnly			:= 	FALSE,
		FirstPosition		:= 	0.0,
		LastPosition		:= 	0.0,
		Options				:= 	,
		Done				=> 	,
		Busy				=> 	,
		Error				=> 	,
		ErrorID				=> 	,
		RecordedPosition	=>	fPositionTouch);

(* End *)

END_PROGRAM

// ---- POUs/TwinSAFE/TwinSAFE.TcPOU
PROGRAM TwinSAFE
(*******************************************************************************************************
Description			:	Exsample handling of the TwinSAFE part
Date 				:	04.04.2016
********************************************************************************************************)
VAR

	bTsReadyToReset							:BOOL;
	tBlinkerDelay							:TIME;
	fbBlinker								:FB_Blinker;

	fbSafeGroup1 							:FB_TwinSafeGroup;				(* TwinSAFE group 1 diagnosis *)

	fbSafeFB_1_Group1 						:FB_TwinSafeFB;					(* TwinSAFE function block 1 diagnosis group 1 *)
	fbSafeFB_2_Group1 						:FB_TwinSafeFB;					(* TwinSAFE function block 2 diagnosis group 1 *)
	fbSafeFB_3_Group1 						:FB_TwinSafeFB;					(* TwinSAFE function block 3 diagnosis group 1 *)

	fbSafeConnectionEL1904_1_Group1			:FB_TwinSafeConnectionEL1904;	(* TwinSAFE connection and module diagnosis EL1904-1 group 1 *)
	fbSafeConnectionEL1904_2_Group1			:FB_TwinSafeConnectionEL1904;	(* TwinSAFE connection and module diagnosis EL1904-2 group 1 *)
	fbSafeConnectionEL2904_1_Group1			:FB_TwinSafeConnectionEL2904;	(* TwinSAFE connection and module diagnosis EL2904-1 group 1 *)
	fbSafeConnectionAX5805_1_Group1			:FB_TwinSafeConnectionAX5805;	(* TwinSAFE connection and module diagnosis AX5805-1 group 1 *)

END_VAR
(*******************************************************************************************************
Version/Date:	
V1.0.0 / 03.05.2016 / 
********************************************************************************************************)
(* End *)

(* TwinSAFE sample *)

(* THIS CODE IS ONLY AN EXAMPLE - YOU HAVE TO CHECK APTITUDE FOR YOUR APPLICATION *)

	(* TwinSAFE group diagnosis *)
		fbSafeGroup1(
			bRun	:= TRUE,
			bErrAck	:= bSwitchS31,
			sName	:= 'Group 1');
	
		fbSafeGroup1.bFbErr;
		fbSafeGroup1.bComErr;
		fbSafeGroup1.bOutErr;
		
				
	(* TwinSAFE function block diagnosis *)
		fbSafeFB_1_Group1(
			sName	:=	'FBEStop1',					(* Name in the TwinSAFE drawing *)
			eFBType	:=	E_TsFbType.FB_TYPE_ESTOP, 	(* FB-Type *)
			nFbId	:=	1);							(* Module number in the TwinSAFE drawing *)

		fbSafeFB_2_Group1(
			sName	:=	'FBMon1',					(* Name in the TwinSAFE drawing *)
			eFBType	:=	E_TsFbType.FB_TYPE_MON,		(* FB-Type *)
			nFbId	:=	3);							(* Module number in the TwinSAFE drawing *)

		fbSafeFB_3_Group1(
			sName	:=	'FBEStop2',					(* Name in the TwinSAFE drawing *)
			eFBType	:=	E_TsFbType.FB_TYPE_ESTOP,	(* FB-Type *)
			nFbId	:=	5);							(* Module number in the TwinSAFE drawing *)


	(* TwinSAFE connection and module diagnostic *)
		fbSafeConnectionEL1904_1_Group1(
			tCoEReadCycle 	:= T#2S);	
			
		fbSafeConnectionEL1904_2_Group1(
			tCoEReadCycle 	:= T#2S);	

		fbSafeConnectionEL2904_1_Group1(
			tCoEReadCycle 	:= T#2S); 	

		fbSafeConnectionAX5805_1_Group1(
			tCoEReadCycle	:= T#2S);
			
			
	(* Ready to reset - bLedH31 *)
		IF fbSafeConnectionEL1904_1_Group1.bChannel1			(* Switch S30 *)
		AND fbSafeConnectionEL1904_1_Group1.bChannel2
		AND ((fbSafeConnectionEL1904_2_Group1.bChannel1			(* Switch S32 *)
			AND fbSafeConnectionEL1904_2_Group1.bChannel2)
		OR (NOT fbSafeConnectionEL1904_2_Group1.bChannel3		(* Switch S33 *)
			AND fbSafeConnectionEL1904_2_Group1.bChannel4))
		AND fbSafeConnectionEL1904_1_Group1.nEcSlaveState.3		(* EterCAT Slave in OP *)	
		AND fbSafeConnectionEL1904_2_Group1.nEcSlaveState.3		(* EterCAT Slave in OP *)
		AND fbSafeConnectionEL2904_1_Group1.nEcSlaveState.3		(* EterCAT Slave in OP *)
		THEN
			bTsReadyToReset := TRUE;
		ELSE
			bTsReadyToReset := FALSE;
		END_IF

		IF  fbSafeGroup1.sState <> 'RUN'
			OR fbSafeFB_1_Group1.sState <> 'RUN'
		THEN
			(* Blinker delay wait reset group or Estop *)
			tBlinkerDelay := T#750MS;
		ELSE
			(* Blinker delay wait reset STO *)
			tBlinkerDelay := T#250MS;
		END_IF

		IF fbSafeFB_3_Group1.sState = 'RUN'	
		THEN
			(* Estop and STO run *)
			fbBlinker(bStart := FALSE);
			bLedH31 := TRUE;
		ELSE
			(* Estop or STO not run *)
			fbBlinker(
				bStart			:= 	bTsReadyToReset,
				tTurnOnDelay	:= 	tBlinkerDelay,
				tTurnOffDelay	:= 	tBlinkerDelay,
				bLed			=>	bLedH31);
		END_IF

		bLedH32 := (NOT fbSafeConnectionEL1904_2_Group1.bChannel1
						OR NOT fbSafeConnectionEL1904_2_Group1.bChannel2)
							AND fbSafeConnectionEL1904_2_Group1.nEcSlaveState.3;

		bLedH33 := (NOT fbSafeConnectionEL1904_2_Group1.bChannel3
						AND fbSafeConnectionEL1904_2_Group1.bChannel4)
							AND fbSafeConnectionEL1904_2_Group1.nEcSlaveState.3;
		
(* End *)

END_PROGRAM

// ---- POUs/TwinSAFE/Components/FB_TwinSafeGroup.TcPOU
FUNCTION_BLOCK FB_TwinSafeGroup
(*******************************************************************************************************
Description			:	Entries of the status and diagnostic TwinSAFE groups
ocumentation 		:	TwinSAFE-Logik-FB TwinCAT function blocks for TwinSAFE logic terminals
Supported hardware	: 	KL6904 / EL6900
Version/Date 		:	V3.1.0/26.10.2016
********************************************************************************************************)
VAR_INPUT

	bRun							AT %Q*	:BOOL;				(* TwinSAFE group run - linked with the associated TwinSAFE Group in the TwinSAFE projekt *)
	bErrAck							AT %Q*	:BOOL;				(* TwinSAFE group error acknowledge - linked with the associated TwinSAFE Group in the TwinSAFE projekt *)
	sName									:STRING;			(* TwinSAFE group name *)

END_VAR
VAR_OUTPUT

	stInfoData						AT %I*	:ST_TsGroupInfo;	(* TwinSAFE Group Info Data *)
	bFbErr							AT %I*	:BOOL;				(* TwinSAFE group function block error - linked with the associated TwinSAFE Group in the TwinSAFE projekt *)
	bComErr							AT %I*	:BOOL;				(* TwinSAFE group communication error - linked with the associated TwinSAFE Group in the TwinSAFE projekt *)
	bOutErr							AT %I*	:BOOL;				(* TwinSAFE group output error - linked with the associated TwinSAFE Group in the TwinSAFE projekt *)
	sState									:STRING;
	
END_VAR
VAR
END_VAR
(* End *)

(* TwinSAFE group status and diagnostic *)

(* THIS CODE IS ONLY AN EXAMPLE - YOU HAVE TO CHECK APTITUDE FOR YOUR APPLICATION *)

	CASE stInfoData.nState OF
		1:	sState := 'RUN';
		2:	sState := 'STOP';
		3:	sState := 'SAFE';
		4:	sState := 'ERROR';
		5:	sState := 'RESET';
	ELSE
		sState := 'undefined';
	END_CASE

(* End *)

END_FUNCTION_BLOCK

// ---- POUs/TwinSAFE/Components/FB_TwinSafeFB.TcPOU
FUNCTION_BLOCK FB_TwinSafeFB
(*******************************************************************************************************
Description			:	Entries of the status and diagnostic TwinSAFE function blocks
Documentation 		:	TwinSAFE-Logik-FB TwinCAT function blocks for TwinSAFE logic terminals
Supported hardware	: 	KL6904 / EL6900 / EL6910 / EJ6910 / EK1960
Version/Date 		:	V3.1.0/26.10.2016
********************************************************************************************************)
VAR_INPUT

	sName									:STRING;		(* TwinSAFE function block Name in the TwinSAFE project *)
	eFBType									:E_TsFbType;	(* TwinSAFE function block type in the TwinSAFE project *)
	nFbId									:UINT;			(* TwinSAFE function block ID in the TwinSAFE project *)

END_VAR
VAR_OUTPUT
	
	stInfoData						AT%I* 	:ST_TsFbInfo;	(* Function Block Info Data *)
	sType									:STRING;
	sState									:STRING;
	sDiag									:STRING;

END_VAR
VAR
END_VAR
(* End *)

(* TwinSAFE function block status and diagnosis *)	

(* THIS CODE IS ONLY AN EXAMPLE - YOU HAVE TO CHECK APTITUDE FOR YOUR APPLICATION *)

	CASE eFBType OF
		
		FB_TYPE_AND					:	(* TwinSAFE function block - AND *)

			sType := 'AND';
			
			CASE stInfoData.nState OF
				1:		sState := 'RUN';	
				2:		sState := 'STOP';	
				3:		sState := 'SAFE';	
			ELSE 
				sState := 'undefined';
			END_CASE
			
			sDiag := 'NOT IN USE';


		FB_TYPE_OR					:	(* TwinSAFE function block - OR *)

			sType := 'OR';
			
			CASE stInfoData.nState OF
				1:		sState := 'RUN';	
				2:		sState := 'STOP';	
				3:		sState := 'SAFE';	
			ELSE 	
				sState := 'undefined';
			END_CASE

			sDiag := 'NOT IN USE';

			
		FB_TYPE_OPMODE				:	(* TwinSAFE function block - OPMODE *)

			sType := 'OPMODE';
			
			CASE stInfoData.nState OF
				1:		sState := 'RUN';	
				2:		sState := 'STOP';	
				3:		sState := 'SAFE';	
				4:		sState := 'ERROR';	
				5:		sState := 'RESET';	
				6:		sState := 'START';	
			ELSE 
				sState := 'undefined';
			END_CASE
			
			CASE stInfoData.nDiag OF
				0:	sDiag := 'No error';		
				1:	sDiag := 'Discrepancy monitoring error';		
			ELSE 
				sDiag := 'undefined';
			END_CASE


		FB_TYPE_ESTOP				:	(* TwinSAFE function block - ESTOP *)

			sType := 'ESTOP';
			
			CASE stInfoData.nState OF
				1:		sState := 'RUN';	
				2:		sState := 'STOP';	
				3:		sState := 'SAFE';	
				4:		sState := 'ERROR';	
				5:		sState := 'RESET';	
				6:		sState := 'START';	
				8:		sState := 'DELAYOUT';	
			ELSE 
				sState := 'undefined';
			END_CASE

			
			sDiag := '';
			
			CASE TO_WORD(stInfoData.nDiag) AND 16#00FF OF
				1:		sDiag := 'Discrepancy error input group 1';
				2:		sDiag := 'Discrepancy error input group 2';
				4:		sDiag := 'Discrepancy error input group 3';
				8:		sDiag := 'Discrepancy error input group 4';
				16:		sDiag := 'EDM monitoring error EDM1';
				32:		sDiag := 'EDM monitoring error EDM2';
			END_CASE

			CASE TO_WORD(stInfoData.nDiag) AND 16#FF00 OF
				256:	sDiag := CONCAT(sDiag, ' - option "SAFE Inputs after Disc Error" aktiv');
				512:	sDiag := CONCAT(sDiag, ' - option "SAFE Inputs after Disc Error" aktiv');
				1024:	sDiag := CONCAT(sDiag, ' - option "SAFE Inputs after Disc Error" aktiv');
				2048:	sDiag := CONCAT(sDiag, ' - option "SAFE Inputs after Disc Error" aktiv');
			END_CASE
				
			IF stInfoData.nDiag = 0
			THEN
				sDiag := 'No error';
			ELSIF sDiag = ''
			THEN
				sDiag := 'undefined';		
			END_IF

			
		FB_TYPE_MON					:	(* TwinSAFE function block - MON *)

			sType := 'MON';
			
			CASE stInfoData.nState OF
				1:		sState := 'RUN';	
				2:		sState := 'STOP';	
				3:		sState := 'SAFE';	
				4:		sState := 'ERROR';	
				5:		sState := 'RESET';	
				6:		sState := 'START';	
				7:		sState := 'ERRORDELAY';	
				8:		sState := 'DELAYOUT';	
				9:		sState := 'FUNCTEST';	
			ELSE 
				sState := 'undefined';
			END_CASE
			
			CASE stInfoData.nDiag OF
				0:		sDiag := 'No error';		
				1:		sDiag := 'Discrepancy error input group 1';	
				2:		sDiag := 'Discrepancy error input group 1';		
				4:		sDiag := 'Discrepancy error in Secure input group';	
				16:		sDiag := 'EDM monitoring error EDM1';	
				32:		sDiag := 'EDM monitoring error EDM2';	
			ELSE 
				sDiag := 'undefined';
			END_CASE


		FB_TYPE_DECOUPLER			:	(* TwinSAFE function block - DECOUPLER *)

			sType := 'DECOUPLER';
			
			CASE stInfoData.nState OF
				1:		sState := 'RUN';	
				2:		sState := 'STOP';	
			ELSE 
				sState := 'undefined';
			END_CASE

			sDiag := 'NOT IN USE';

			
		FB_TYPE_TWOHAND				:	(* TwinSAFE function block - TWOHAND *)

			sType := 'TWO-HAND';
			
			CASE stInfoData.nState OF
				1:		sState := 'RUN';	
				2:		sState := 'STOP';	
				3:		sState := 'SAFE';	
				4:		sState := 'ERROR';		
				5:		sState := 'RESET';	
				6:		sState := 'START';	
				11:		sState := '1BUTTON';	
				12:		sState := '2BUTTON';	
				13:		sState := 'RELEASE';	
			ELSE 
				sState := 'undefined';
			END_CASE
			
			CASE stInfoData.nDiag OF
				0:		sDiag := 'No error';		
				1:		sDiag := 'Discrepancy error input group 1';	
				2:		sDiag := 'Discrepancy error input group 1';	
				4:		sDiag := 'Discrepancy error between the two input groups';	
				64:		sDiag := 'Two-hand error';	
			ELSE 
				sDiag := 'undefined';
			END_CASE

	
		FB_TYPE_MUTING				:	(* TwinSAFE function block - MUTING  *)

			sType := 'MUTING';
			
			CASE stInfoData.nState OF
				1:		sState := 'RUN';	
				2:		sState := 'STOP';	
				3:		sState := 'SAFE';	
				4:		sState := 'ERROR';	
				5:		sState := 'RESET';	
				8:		sState := 'DELAYOUT';	
				9:		sState := 'MUTING1';	
				10:		sState := 'MUTING2';	
				11:		sState := 'MUTING3';	
				12:		sState := 'MUTING4';	
				13:		sState := 'MUTING5';	
				14:		sState := 'MUTING6';	
				15:		sState := 'MUTING7';	
				16:		sState := 'MUTING8';	
				17:		sState := 'MUTING9';	
			ELSE 
				sState := 'undefined';
			END_CASE
			
			CASE stInfoData.nDiag OF
				0:		sDiag := 'No error';		
				1:		sDiag := 'Discrepancy error in muting input group 1';	
				2:		sDiag := 'Discrepancy error in the OSSD input group';	
				4:		sDiag := 'Discrepancy error in muting input group 2';	
				16:		sDiag := 'EDM monitoring error EDM1';	
				32:		sDiag := 'EDM monitoring error EDM2';	
				64:		sDiag := 'Muting sequence was violated';	
				128:	sDiag := 'Maximum muting time was exceeded';	
			ELSE 
				sDiag := 'undefined';
			END_CASE

		
		FB_TYPE_EDM					:	(* TwinSAFE function block - EDM *)

			sType := 'EDM';
			
			CASE stInfoData.nState OF
				2:		sState := 'STOP';	
				4:		sState := 'ERROR';	
				5:		sState := 'RESET';	
				14:		sState := 'MON_OFF';	
				15:		sState := 'MON_ON';	
			ELSE 
				sState := 'undefined';
			END_CASE
			
			CASE stInfoData.nDiag OF
				0:		sDiag := 'No error';		
				1:		sDiag := 'Switch-OFF timer elapsed';	
				2:		sDiag := 'Switch-ON timer elapsed';	
			ELSE 
				sDiag := 'undefined';
			END_CASE

			
		FB_TYPE_RS					:	(* TwinSAFE function block - RS *)

			sType := 'RS';

			CASE stInfoData.nState OF
				2:		sState := 'STOP';	
				3:		sState := 'SAFE';	
				9:		sState := 'SET';	
			ELSE 
				sState := 'undefined';
			END_CASE

			sDiag := 'NOT IN USE';


		FB_TYPE_SR					:	(* TwinSAFE function block - SR *)

			sType := 'SR';
			
			CASE stInfoData.nState OF
				2:		sState := 'STOP';	
				3:		sState := 'SAFE';	
				9:		sState := 'SET';	
			ELSE 
				sState := 'undefined';
			END_CASE
			
			sDiag := 'NOT IN USE';
	

		FB_TYPE_TON					:	(* TwinSAFE function block - TON *)

			sType := 'TON';
			
			CASE stInfoData.nState OF
				1:		sState := 'RUN';	
				2:		sState := 'STOP';	
				3:		sState := 'SAFE';	
				9:		sState := 'DELAY_IN';	
			ELSE 
				sState := 'undefined';
			END_CASE

			sDiag := 'NOT IN USE';


		FB_TYPE_TOF					:	(* TwinSAFE function block - TOF *)

			sType := 'TOF';
			
			CASE stInfoData.nState OF
				1:		sState := 'RUN';	
				2:		sState := 'STOP';	
				3:		sState := 'SAFE';	
				8:		sState := 'DELAY_OUT';	
			ELSE 
				sState := 'undefined';
			END_CASE

			sDiag := 'NOT IN USE';


		FB_TYPE_CONSHUT				:	(* TwinSAFE function block - CONNECTION SHUTDOWN *)

			sType := 'ConShut';
			
			CASE stInfoData.nState OF
				2:		sState := 'STOP';	
				3:		sState := 'SAFE';	
				4:		sState := 'ERROR';	
				5:		sState := 'RESET';	
				10:		sState := 'ACTIVE';	
				11:		sState := 'DEACTIVE';	
			ELSE 
				sState := 'undefined';
			END_CASE
			
			CASE stInfoData.nDiag OF
				0:		sDiag := 'No error';		
				1:		sDiag := 'Discrepancy error input group 1';	
			ELSE 
				sDiag := 'undefined';
			END_CASE
			
			
		FB_TYPE_ADD					:	(* TwinSAFE function block - ADD *)

			sType := 'ADD';
			
			CASE stInfoData.nState OF
				0:		sState := 'not in use';	
				1:		sState := 'RUN';	
				2:		sState := 'STOP';	
				3:		sState := 'not in use';	
				4:		sState := 'ERROR';	
				5:		sState := 'RESET';	
			ELSE 
				sState := 'undefined';
			END_CASE

			CASE stInfoData.nDiag OF
				0:		sDiag := 'AnalogOut is correct';		
				1:		sDiag := 'AnalogOut has an underflow';	
				2:		sDiag := 'AnalogOut has an overflow';	
			ELSE 
				sDiag := 'undefined';
			END_CASE
			
			
		FB_TYPE_SUB					:	(* TwinSAFE function block - SUB *)

			sType := 'SUB';
			
			CASE stInfoData.nState OF
				0:		sState := 'not in use';	
				1:		sState := 'RUN';	
				2:		sState := 'STOP';	
				3:		sState := 'not in use';	
				4:		sState := 'ERROR';	
				5:		sState := 'RESET';	
			ELSE 
				sState := 'undefined';
			END_CASE

			CASE stInfoData.nDiag OF
				0:		sDiag := 'AnalogOut is correct';		
				1:		sDiag := 'AnalogOut has an underflow';	
				2:		sDiag := 'AnalogOut has an overflow';	
			ELSE 
				sDiag := 'undefined';
			END_CASE

			
		FB_TYPE_MUL					:	(* TwinSAFE function block - MUL *)

			sType := 'MUL';
			
			CASE stInfoData.nState OF
				0:		sState := 'not in use';	
				1:		sState := 'RUN';	
				2:		sState := 'STOP';	
				3:		sState := 'not in use';	
				4:		sState := 'ERROR';	
				5:		sState := 'RESET';	
			ELSE 
				sState := 'undefined';
			END_CASE

			CASE stInfoData.nDiag OF
				0:		sDiag := 'AnalogOut is correct';		
				1:		sDiag := 'AnalogOut has an underflow';	
				2:		sDiag := 'AnalogOut has an overflow';	
			ELSE 
				sDiag := 'undefined';
			END_CASE

			
		FB_TYPE_DIV					:	(* TwinSAFE function block - DIV *)

			sType := 'DIV';
			
			CASE stInfoData.nState OF
				0:		sState := 'not in use';	
				1:		sState := 'RUN';	
				2:		sState := 'STOP';	
				3:		sState := 'not in use';	
				4:		sState := 'ERROR';	
				5:		sState := 'RESET';	
			ELSE 
				sState := 'undefined';
			END_CASE

			CASE stInfoData.nDiag OF
				0:		sDiag := 'AnalogOut is correct';		
				1:		sDiag := 'AnalogOut has an underflow';	
				2:		sDiag := 'AnalogOut has an overflow';	
			ELSE 
				sDiag := 'undefined';
			END_CASE


		FB_TYPE_COMPARE				:	(* TwinSAFE function block - COMPARE *)

			sType := 'COMPARE';
			
			CASE stInfoData.nState OF
				1:		sState := 'RUN';	
				2:		sState := 'STOP';	
				3:		sState := 'SAFE';	
				4:		sState := 'ERROR';	
				5:		sState := 'RESET';	
				8:		sState := 'DELAYOUT';	
			ELSE 
				sState := 'undefined';
			END_CASE

			CASE stInfoData.nDiag OF
				0:		sDiag := 'CompOut is correct';		
				1:		sDiag := 'The output CompOut has an underflow';	
				2:		sDiag := 'The output CompOut has an overflow';	
			ELSE 
				sDiag := 'undefined';
			END_CASE
			
			
		FB_TYPE_LIMIT				:	(* TwinSAFE function block - LIMIT *)

			sType := 'LIMIT';
			
			CASE stInfoData.nState OF
				1:		sState := 'RUN';	
				2:		sState := 'STOP';	
				3:		sState := 'SAFE';	
				4:		sState := 'ERROR';	
				5:		sState := 'RESET';	
			ELSE 
				sState := 'undefined';
			END_CASE

			CASE stInfoData.nDiag OF
				0:		sDiag := 'No error';		
				1:		sDiag := 'MinValue > MaxValue';	
			ELSE 
				sDiag := 'undefined';
			END_CASE
			
			
		FB_TYPE_COUNTER				:	(* TwinSAFE function block - COUNTER *)

			sType := 'COUNTER';
			
			CASE stInfoData.nState OF
				1:		sState := 'RUN';	
				2:		sState := 'STOP';	
				4:		sState := 'ERROR';	
				5:		sState := 'RESET';	
			ELSE 
				sState := 'undefined';
			END_CASE

			CASE stInfoData.nDiag OF
				0:		sDiag := 'No error';		
				1:		sDiag := 'ActValue has an underflow';	
				2:		sDiag := 'ActValue has an overflow';	
			ELSE 
				sDiag := 'undefined';
			END_CASE


		FB_TYPE_SCALE				:	(* TwinSAFE function block - SCALE *)

			sType := 'SCALE';
			
			CASE stInfoData.nState OF
				1:		sState := 'RUN';	
				2:		sState := 'STOP';	
				4:		sState := 'ERROR';	
				5:		sState := 'RESET';	
			ELSE 
				sState := 'undefined';
			END_CASE

			CASE stInfoData.nDiag OF
				0:		sDiag := 'No error';		
				1:		sDiag := 'AnalogOut has an underflow';	
				2:		sDiag := 'AnalogOut has an overflow';	
				3:		sDiag := 'A 32-bit overflow occurs during the multiplication';	
				4:		sDiag := 'A 32-bit overflow occurs during by rounding up at the division ';	
			ELSE 
				sDiag := 'undefined';
			END_CASE


		FB_TYPE_SPEED				:	(* TwinSAFE function block - SPEED *)

			sType := 'SPEED';
			
			CASE stInfoData.nState OF
				1:		sState := 'RUN';	
				2:		sState := 'STOP';	
				4:		sState := 'ERROR';	
				5:		sState := 'RESET';	
			ELSE 
				sState := 'undefined';
			END_CASE

			CASE stInfoData.nDiag OF
				0:		sDiag := 'No error';		
				1:		sDiag := 'The output Speed has an underflow';	
				2:		sDiag := 'The output Speed has an overflow';	
			ELSE 
				sDiag := 'undefined';
			END_CASE


		FB_TYPE_LOADSENSING			:	(* TwinSAFE function block - LOAD SENSING *)

			sType := 'LOADSENSING';
			
			CASE stInfoData.nState OF
				1:		sState := 'RUN';	
				2:		sState := 'STOP';	
				3:		sState := 'SAFE';	
				16:		sState := 'INACTIVE';	
				17:		sState := 'WARNING';	
			ELSE 
				sState := 'undefined';
			END_CASE

			sDiag := 'NOT IN USE';


		FB_TYPE_CAMMONITOR			:	(* TwinSAFE function block - CAM MONITOR *)

			sType := 'CAMMONITOR';
			
			CASE stInfoData.nState OF
				1:		sState := 'RUN';	
				2:		sState := 'STOP';	
				3:		sState := 'SAFE';	
				4:		sState := 'ERROR';	
				5:		sState := 'RESET';	
				6:		sState := 'START';	
				15:		sState := 'WAIT-FOR-RESET';	
				16:		sState := 'MOVE-STOP';	
				17:		sState := 'MOVE-START';	
				18:		sState := 'MOVE-DOWN';	
				19:		sState := 'MOVE-UP';	
				20:		sState := 'MOVE-TDC';	
				32:		sState := 'MOVE-DOWN-CLOCKWISE';	
				33:		sState := 'MOVE-UP-CLOCKWISE';	
				34:		sState := 'MOVE-UP-TDC1';	
				35:		sState := 'MOVE-STOP-TDC1';	
				36:		sState := 'MOVE-START-TDC1';	
				37:		sState := 'MOVE-DOWN-CONTRA-CLOCKWISE';	
				38:		sState := 'MOVE-UP-CONTRA-CLOCKWISE';	
				39:		sState := 'MOVE-UP-TDC2';	
				40:		sState := 'MOVE-STOP-TDC2';	
				41:		sState := 'MOVE-START-TDC2';	
			ELSE 
				sState := 'undefined';
			END_CASE

			sDiag := 'NOT IN USE';


		FB_TYPE_SLI					:	(* TwinSAFE function block - SLI *)

			sType := 'SLI';
			
			CASE stInfoData.nState OF
				1:		sState := 'RUN';	
				2:		sState := 'STOP';	
				3:		sState := 'SAFE';	
				4:		sState := 'ERROR';	
				5:		sState := 'RESET';	
			ELSE 
				sState := 'undefined';
			END_CASE

			CASE stInfoData.nDiag OF
				0:		sDiag := 'No error';		
				1:		sDiag := 'Underflow (PositionDiff < -NegLimit)';		
				2:		sDiag := 'Overflow (PositionDiff > PosLimit)';		
			ELSE 
				sDiag := 'undefined';
			END_CASE


		FB_TYPE_ENVELOPE			:	(* TwinSAFE function block - ENVELOPE *)

			sType := 'ENVELOPE';
			
			CASE stInfoData.nState OF
				1:		sState := 'RUN';	
				2:		sState := 'STOP';	
				3:		sState := 'SAFE';	
				4:		sState := 'ERROR';	
				5:		sState := 'RESET';	
				8:		sState := 'DELAYOUT';	
				9:		sState := 'MONITOR';	
			ELSE 
				sState := 'undefined';
			END_CASE

			CASE stInfoData.nDiag OF
				0:		sDiag := 'No error';		
				1:		sDiag := 'Underflow (InValue below the envelope curve)';		
				2:		sDiag := 'Overflow (InValue above the envelope curve)';		
				3:		sDiag := 'InValue error';		
				4:		sDiag := 'Max time expired)';		
			ELSE 
				sDiag := 'undefined';
			END_CASE


		FB_TYPE_VIOLATIONCOUNTER	:	(* TwinSAFE function block - VIOLATION COUNTER *)

			sType := 'VIOLATIONCOUNTER';
			
			CASE stInfoData.nState OF
				1:		sState := 'RUN';	
				2:		sState := 'STOP';	
				3:		sState := 'SAFE';	
				6:		sState := 'START';	
			ELSE 
				sState := 'undefined';
			END_CASE

			sDiag := 'NOT IN USE';


	ELSE
		
		sType  := 'UNKNOWN FB';
		sState := 'UNKNOWN';
		sDiag  := 'UNKNOWN';

	END_CASE
	
	sType := CONCAT(' : ', sType);
	sType := CONCAT(UINT_TO_STRING(nFbId), sType);
	sType := CONCAT('FB ', sType);
	
(* End *)

END_FUNCTION_BLOCK

// ---- POUs/TwinSAFE/Components/FB_TwinSafeConnectionEL1904.TcPOU
FUNCTION_BLOCK FB_TwinSafeConnectionEL1904
(*******************************************************************************************************
Description			:	Evaluate a TwinSAFE connection status and diagnosis to an EtherCAT terminal
Supported terminals : 	EL1904
Documentation 		:	EL1904 TwinSAFE input terminal with 4 fail-safe inputs
Version/Date 		:	V1.5.2/02.10.2015
Required libraries 	: 	TcSystem.lib (Tc2_System), TcEtherCAT.lib (Tc2_EtherCAT)
********************************************************************************************************)
VAR_INPUT
	
	tCoEReadCycle							:TIME 	:= T#0MS;				(* Read cycle CoE-Data, e.g. temperature *)

END_VAR
VAR_OUTPUT

	stInfoData						AT %I*	:ST_TsConnectionInfo1Byte;		(* EL6900 \ Connection Info Data \ Message_X Info Data*)
	nEcSlaveState					AT %I*	:UINT ;							(* EL1904 \ InfoData \ State *)
	stEcAdsAddr						AT %I*	:ST_AdsAddr;					(* EL1904 \ InfoData \ AdsAddr *)

(* act_EcSlaveIdentify *)
	sEcSlaveType							:STRING(15);
	sEcSlaveName							:STRING(31) := '';
	bSlaveIdentify							:BOOL;
	bSlaveTypeError							:BOOL;
	
(* act_Signals *)
	bChannel1								:BOOL;							
	bChannel2								:BOOL;
	bChannel3								:BOOL;
	bChannel4								:BOOL;

(* act_ConnectionState *)
	sState									:STRING;
	
(* act_ConnectionDiag *)
	sDiag									:STRING;
	sFault									:STRING;						(* FailSafe Error (Hardware)*)
	bError									:BOOL;							(* TwinSAFE-Error *)
	
(* act_ReadDiagObjects *)
	stSlaveTemp								:ST_TsSlave2Temp;
	bTempWarning							:BOOL;							(* Temperature warning: T1, T2 *)
	stTsDiagObjectsBitsEL1904				:ST_TsDiagObjectsBitsEL1904;

END_VAR
VAR

(* act_ConnectionDiag *)
	nDiag0_3								:BYTE;

(* act_ReadDiagObjects *)
	eReadDiagObjState						:E_TsCycleDiagObj;
	eReadDiagObjErrStep						:E_TsCycleDiagObj := E_TsCycleDiagObj.eCycleDiagObj_NoError;
	bReadDiagObjError						:BOOL;							(* Error in the diagnosis objects read cycle *)  
	bReadDiagObjReset						:BOOL;							(* Reset the diagnosis objects read cycle error *)
	fbTimer									:TON;
	fbEcCoeSdoRead							:FB_EcCoESdoReadEx;
	stDiagObjects							:ST_TsDiagObjectsEL1904;

(* act_EcSlaveIdentify *)
	fbEcGetSlaveName						:FB_EcGetSlaveName;

END_VAR
VAR CONSTANT
	
(* act_ReadDiagObjects *)
	nWarningLevelTemp1						:INT	:= 85;					(* Temperature 1 warning level [°C] *)
	nWarningLevelTemp2						:INT	:= 85;					(* Temperature 2 warning level [°C] *)

END_VAR
(* End *)

(* Function Block TwinSAFE connection status and diagnosis for EL1904 Terminals *)

(* THIS CODE IS ONLY AN EXAMPLE - YOU HAVE TO CHECK APTITUDE FOR YOUR APPLICATION *)

	(* Identify the EtherCAT slave *)
		act_EcSlaveIdentify();

	(* Evaluate the connection state *)
		act_ConnectionState();
	
	(* Evaluate the connection diagnosis *)
		act_ConnectionDiag();
	
	(* Evaluate the EL1904 input signals *)
		act_Signals();
	
	(* Evaluate the Terminal temperatures and diagnostic objects *)
		IF bSlaveIdentify
		THEN
			act_ReadDiagObjects();
		ELSE
			eReadDiagObjState := E_TsCycleDiagObj.eCycleDiagObj_Init;
		END_IF
		
(* End *)

ACTION act_ConnectionDiag:
(* Evaluate the connection diagnosis *)

	(* Evaluate Bit 0..3 *)
	nDiag0_3 := USINT_TO_BYTE(stInfoData.nDiag) AND 16#0F;

	CASE nDiag0_3 OF
		0:		sDiag := 'No error';
		1:		sDiag := 'Invalid command';
		2:		sDiag := 'Unknown command';
		3:		sDiag := 'Invalid connection ID';
		4:		sDiag := 'Invalid CRC';
		5:		sDiag := 'Watchdog time elapsed';
		6:		sDiag := 'Invalid FSOE address';
		7:		sDiag := 'Invalid data';
		8:		sDiag := 'Invalid communication parameter length';
		9:		sDiag := 'Invalid communication parameters';
		10:		sDiag := 'Invalid user parameter length';
		11:		sDiag := 'Invalid user parameter';
		12:		sDiag := 'FSoE master reset';
		13:		sDiag := 'Module err detected on slave, with option "Module error is ComError" activated';
		14:		sDiag := 'Module err detected on EL290x, with option "Error acknowledge active" activated';
		15:		sDiag := 'Slave not yet started, or unexpected error argument';
	END_CASE

	(* Evaluate Bit 4..7 *)
	sFault:='';

	IF stInfoData.nDiag.4 
	THEN
		sFault	:= 'FSoE slave error detected - '; 
	END_IF

	IF stInfoData.nDiag.5 
	THEN
		sFault	:= concat(sFault,'FSoE slave reports Failsafe Value active - ');
	END_IF

	IF stInfoData.nDiag.6 
	THEN
		sFault	:= concat(sFault,'StartUp - ');
	END_IF

	IF stInfoData.nDiag.7 
	THEN
		sFault	:= concat(sFault, 'FSoE master reports Failsafe Value active');
	END_IF
		
	(* Error *)
	bError := stInfoData.nDiag <> 0;

(* End *)
END_ACTION

ACTION act_ConnectionState:
(* Evaluate the connection state *)

	CASE stInfoData.nState OF
		100:	sState := 'Reset state';
		101:	sState := 'Session state';
		102:	sState := 'Connection state';
		103:	sState := 'Parameter state';
		104:	sState := 'Data state';
		105:	sState := 'Shutdown state';
	ELSE
		sState := 'unknown';
	END_CASE
	
(* End *)
END_ACTION

ACTION act_DiagObjectsBits:
(* act_TsDiagObjectsBits *)

	stTsDiagObjectsBitsEL1904.bErrInput1		 			 := stDiagObjects.nSensorTestError.0;
	stTsDiagObjectsBitsEL1904.bErrInput2		 			 := stDiagObjects.nSensorTestError.1;
	stTsDiagObjectsBitsEL1904.bErrInput3		 			 := stDiagObjects.nSensorTestError.2;
	stTsDiagObjectsBitsEL1904.bErrInput4		 			 := stDiagObjects.nSensorTestError.1;
	
	stTsDiagObjectsBitsEL1904.bErrFirstInputPair 			 := stDiagObjects.nDuringTwoChannelEvaluationError.0;
	stTsDiagObjectsBitsEL1904.bErrSecondInputPair 			 := stDiagObjects.nDuringTwoChannelEvaluationError.1;

	stTsDiagObjectsBitsEL1904.bMatOpModeErrFirstInputPair	 := stDiagObjects.nMatModeInputPairDisagreeError.0 
																	AND stDiagObjects.nMatModeInputPairDisagreeError.1;
	stTsDiagObjectsBitsEL1904.bMatOpModeErrSecondInputPair	 := stDiagObjects.nMatModeInputPairDisagreeError.2 
																	AND stDiagObjects.nMatModeInputPairDisagreeError.3;

	stTsDiagObjectsBitsEL1904.bMatOpModeExtSupplyErrInput1 	 := stDiagObjects.nMatModeExternalSupplyError.0;
	stTsDiagObjectsBitsEL1904.bMatOpModeExtSupplyErrInput2 	 := stDiagObjects.nMatModeExternalSupplyError.1;
	stTsDiagObjectsBitsEL1904.bMatOpModeExtSupplyErrInput3 	 := stDiagObjects.nMatModeExternalSupplyError.2;
	stTsDiagObjectsBitsEL1904.bMatOpModeExtSupplyErrInput4 	 := stDiagObjects.nMatModeExternalSupplyError.3;

(* End *)
END_ACTION

ACTION act_EcSlaveIdentify:
(* Identify the EtherCAT slave *)

	IF NOT nEcSlaveState.3
	THEN
		bSlaveIdentify  := FALSE;
		bSlaveTypeError := FALSE;
		sEcSlaveType    := '';
	END_IF

	IF nEcSlaveState.3
		AND NOT bSlaveIdentify
		AND NOT bSlaveTypeError
 		AND F_CreateAmsNetId(stEcAdsAddr.netId) <> '0.0.0.0.0.0' 
		AND stEcAdsAddr.port <> 0
	THEN

		fbEcCoeSdoRead(
			sNetId			:= 	F_CreateAmsNetId(stEcAdsAddr.netId),
			nSlaveAddr		:= 	stEcAdsAddr.port,
			nSubIndex		:= 	0,
			nIndex			:= 	16#1008,
			pDstBuf			:= 	ADR(sEcSlaveType),
			cbBufLen		:= 	SIZEOF(sEcSlaveType),
			bExecute		:= 	TRUE,
			tTimeout		:= 	DEFAULT_ADS_TIMEOUT);
	

		fbEcGetSlaveName(
			bExecute		:=	TRUE, 
			sNetId			:=	F_CreateAmsNetId(stEcAdsAddr.netId), 
			nSlaveAddr		:=	stEcAdsAddr.port, 
			tTimeout		:=	DEFAULT_ADS_TIMEOUT, 
			bBusy			=>	, 
			sSlaveName		=>	sEcSlaveName, 
			bError			=>	, 
			nErrId			=>	);

		IF NOT fbEcCoeSdoRead.bBusy
			AND NOT fbEcCoeSdoRead.bError
			AND NOT fbEcGetSlaveName.bBusy
			AND NOT fbEcGetSlaveName.bError
		THEN
		
			fbEcCoeSdoRead(bExecute := FALSE); 
			fbEcGetSlaveName(bExecute := FALSE); 

			IF sEcSlaveType = 'EL1904' 
				AND fbEcGetSlaveName.sSlaveName <> ''
			THEN
				bSlaveIdentify := TRUE;
			ELSE
				bSlaveTypeError := TRUE;
			END_IF

		ELSIF NOT fbEcCoeSdoRead.bBusy
			AND fbEcCoeSdoRead.bError
		OR (NOT fbEcGetSlaveName.bBusy
			AND fbEcGetSlaveName.bError)
		THEN
		
			fbEcCoeSdoRead(bExecute := FALSE); 
			fbEcGetSlaveName(bExecute := FALSE); 

		END_IF

	END_IF
	
(* End *)
END_ACTION

ACTION act_ReadDiagObjects:
(* Evaluate the Terminal temperatures and diagnostic objects *)

	CASE eReadDiagObjState OF

		eCycleDiagObj_Init				:	(* Init *)	

			IF nEcSlaveState.3					(* Slave in OP *)
				AND tCoEReadCycle <> T#0MS 		(* tCoEReadCycle <> t#0ms -> Read diagnostic aktiv *)
			THEN
				bReadDiagObjError := FALSE;
				fbEcCoeSdoRead(	bExecute := FALSE);
				fbTimer(IN := FALSE);
				eReadDiagObjState := eCycleDiagObj_ReadTemperature;
			END_IF

			
		eCycleDiagObj_ReadTemperature	:	(* Read temperature *)

			fbEcCoeSdoRead(
				sNetId			:= 	F_CreateAmsNetId(stEcAdsAddr.netId),
				nSlaveAddr		:= 	stEcAdsAddr.port,
				nSubIndex		:= 	1,
				nIndex			:= 	16#FA80,
				pDstBuf			:= 	ADR(stSlaveTemp),
				cbBufLen		:= 	SIZEOF(stSlaveTemp),
				bExecute		:= 	TRUE,
				tTimeout		:= 	DEFAULT_ADS_TIMEOUT,
				bCompleteAccess	:= 	TRUE);

			IF NOT fbEcCoeSdoRead.bBusy 
				AND NOT fbEcCoeSdoRead.bError 
			THEN
				fbEcCoeSdoRead(bExecute := FALSE);
				eReadDiagObjState := eCycleDiagObj_ReadDiag;
			ELSIF NOT fbEcCoeSdoRead.bBusy 
				AND fbEcCoeSdoRead.bError 
			THEN
				eReadDiagObjErrStep := eReadDiagObjState;
				eReadDiagObjState 	:= eCycleDiagObj_Error;
			END_IF

			
		eCycleDiagObj_ReadDiag			:	(* Read diacnostic objects *)

			fbTimer(IN := TRUE, PT := tCoEReadCycle);

			fbEcCoeSdoRead(
				sNetId			:= 	F_CreateAmsNetId(stEcAdsAddr.netId),
				nSlaveAddr		:= 	stEcAdsAddr.port,
				nSubIndex		:= 	1,
				nIndex			:= 	16#800E,
				pDstBuf			:= 	ADR(stDiagObjects),
				cbBufLen		:= 	SIZEOF(stDiagObjects),
				bExecute		:= 	TRUE,
				tTimeout		:= 	DEFAULT_ADS_TIMEOUT,
				bCompleteAccess	:= 	TRUE);

			IF NOT fbEcCoeSdoRead.bBusy 
				AND NOT fbEcCoeSdoRead.bError 
			THEN
				fbEcCoeSdoRead(bExecute := FALSE);
				act_DiagObjectsBits();
				eReadDiagObjState := eCycleDiagObj_ReadDelay;
			ELSIF NOT fbEcCoeSdoRead.bBusy 
				AND fbEcCoeSdoRead.bError 
			THEN
				eReadDiagObjErrStep := eReadDiagObjState;
				eReadDiagObjState 	:= eCycleDiagObj_Error;
			END_IF
				
			
		eCycleDiagObj_ReadDelay		:	(* Read delay *)
			fbTimer(
				IN := TRUE, 
				PT := tCoEReadCycle);

			IF fbTimer.Q 
			THEN
				fbTimer(IN := FALSE); 			
				eReadDiagObjState := eCycleDiagObj_Done;
			END_IF

			
		eCycleDiagObj_Done				:	(* Done *)

			eReadDiagObjState := eCycleDiagObj_Init;

			
		eCycleDiagObj_Error			:	(* Error detected *)

			bReadDiagObjError := TRUE;
		
			IF bReadDiagObjReset
			THEN
				bReadDiagObjError := FALSE;
				fbEcCoeSdoRead(bExecute := FALSE);
				eReadDiagObjErrStep := E_TsCycleDiagObj.eCycleDiagObj_NoError;
				eReadDiagObjState := eCycleDiagObj_Init;
			END_IF

	ELSE
		
		eReadDiagObjState := eCycleDiagObj_Init;
		
	END_CASE

	bTempWarning := stSlaveTemp.nInternalTemperature1 >= nWarningLevelTemp1 
						OR stSlaveTemp.nInternalTemperature2 >= nWarningLevelTemp2;

(* End *)
END_ACTION

ACTION act_Signals:
(* Evaluate the input (EL1904) signals *)

	IF nEcSlaveState.3 (* Slave in operational state *)
	THEN
		(* OP -> transfer the signal states *)
		bChannel1 := stInfoData.nInOutSafeDataByte1.0;
		bChannel2 := stInfoData.nInOutSafeDataByte1.1;
		bChannel3 := stInfoData.nInOutSafeDataByte1.2;
		bChannel4 := stInfoData.nInOutSafeDataByte1.3;
	ELSE
		(* Error -> clear the signal states *)
		bChannel1 := bChannel2 := bChannel3 := bChannel4 := FALSE;
	END_IF

(* End *)
END_ACTION

END_FUNCTION_BLOCK

// ---- POUs/TwinSAFE/Components/FB_EcGetSlaveName.TcPOU
FUNCTION_BLOCK FB_EcGetSlaveName
(*******************************************************************************************************
Title				:	Get EtherCAT slave name
Description			:	Read the EtherCAT slave name from the EtherCAT Master CoE table
Version / Date		:	1.0.0 / 23.05.2016 / created program (Version progress see below)
********************************************************************************************************)
VAR_INPUT

	bExecute                        		:BOOL;							(* The block is activated by a rising edge at this input *)
	sNetId          						:T_AmsNetId;					(* AmsNetId of the EtherCAT master device *)
	nSlaveAddr      						:UINT; 							(* Address of the slave device *)
	tTimeout                        		:TIME := DEFAULT_ADS_TIMEOUT;

END_VAR
VAR_OUTPUT

	bBusy           						:BOOL;							(* This output is set when the function block is activated *)
	sSlaveName         						:STRING[31];					(* Name of this EtherCAT Slave *)
	bError          						:BOOL;
	nErrId          						:UDINT;

END_VAR
VAR

	eStateEcGetSlaveNameSeq					:E_EcGetSlaveName;
	eEcGetSlaveNameErrStep					:E_EcGetSlaveName := eEcGetSlaveName_NoError;

	fbEcGetAllSlaveAddr						:FB_EcGetAllSlaveAddr;
	aAllSlaveAddr							:ARRAY[cMinNumberEcSlaves..cMaxNumberEcSlaves] OF UINT;
	nSlaveAddrIndex							:UINT;
	fbEcCoeSdoRead							:FB_EcCoESdoReadEx;

END_VAR
VAR CONSTANT

	cMinNumberEcSlaves						:UINT := 0;
	cMaxNumberEcSlaves						:UINT := 100;

END_VAR
(*******************************************************************************************************
Version / Date / Description:
1.0.0   / 23.05.2016 / created program
********************************************************************************************************)
(* End *)

(* FB_EcGetSlaveName *)

	CASE eStateEcGetSlaveNameSeq OF 
	
		eEcGetSlaveName_Start				:	(* Waiting for start *)
			
			IF bExecute
			THEN
				bBusy := TRUE;
				eStateEcGetSlaveNameSeq := eEcGetSlaveName_Init;
			END_IF
		
		eEcGetSlaveName_Init				:	(* Initialize functions *)

			fbEcGetAllSlaveAddr(bExecute := FALSE);
			fbEcCoeSdoRead(		bExecute := FALSE);
			
			eStateEcGetSlaveNameSeq := eEcGetSlaveName_ReadAllSlaveAddr;
			
	
		eEcGetSlaveName_ReadAllSlaveAddr	:	(* Read all EtherCAT Slave addresses and find the slave position in the EtherCAT bus *)

			fbEcGetAllSlaveAddr(
				sNetId	 := sNetId, 
				pAddrBuf := ADR(aAllSlaveAddr), 
				cbBufLen := SIZEOF(aAllSlaveAddr), 
				bExecute := TRUE, 
				tTimeout := DEFAULT_ADS_TIMEOUT);

			IF NOT fbEcGetAllSlaveAddr.bBusy
				AND NOT fbEcGetAllSlaveAddr.bError
			THEN
			
				FOR nSlaveAddrIndex := cMinNumberEcSlaves TO cMaxNumberEcSlaves BY 1 DO
					IF nSlaveAddr = aAllSlaveAddr[nSlaveAddrIndex]
					THEN
						EXIT;
					END_IF
				END_FOR

				fbEcGetAllSlaveAddr(bExecute := FALSE);
			
				eStateEcGetSlaveNameSeq := eEcGetSlaveName_ReadSlaveName;
	
			ELSIF NOT fbEcGetAllSlaveAddr.bBusy
				AND fbEcGetAllSlaveAddr.bError
			THEN

				nErrId					:=	fbEcGetAllSlaveAddr.nErrId;
				eEcGetSlaveNameErrStep	:= 	eStateEcGetSlaveNameSeq;
				eStateEcGetSlaveNameSeq := 	eEcGetSlaveName_ErrorStep;
			
			END_IF

		eEcGetSlaveName_ReadSlaveName		:	(* Read the EtherCAT slave name from the EtherCAT master CoE table *)
				
			fbEcCoeSdoRead(
				sNetId		:= sNetId, 
				nSlaveAddr	:= 16#FFFF, 						(* EtherCAT master address = 16#FFFF *)
				nSubIndex	:= 3, 
				nIndex		:= 16#8000 + nSlaveAddrIndex, 
				pDstBuf		:= ADR(sSlaveName), 
				cbBufLen	:= SIZEOF(sSlaveName), 
				bExecute	:= TRUE, 
				tTimeout	:= DEFAULT_ADS_TIMEOUT);	


			IF NOT fbEcCoeSdoRead.bBusy
				AND NOT fbEcCoeSdoRead.bError
			THEN
					
				fbEcCoeSdoRead(bExecute := FALSE);

				eStateEcGetSlaveNameSeq := eEcGetSlaveName_Done;
	
			ELSIF NOT fbEcCoeSdoRead.bBusy
				AND fbEcCoeSdoRead.bError
			THEN
				nErrId					:=	fbEcCoeSdoRead.nErrId;
				eEcGetSlaveNameErrStep	:= 	eStateEcGetSlaveNameSeq;
				eStateEcGetSlaveNameSeq := 	eEcGetSlaveName_ErrorStep;
			
			END_IF


		eEcGetSlaveName_Done				:	(* EtherCAT slave name read done *)

			bBusy := FALSE;

			IF NOT bExecute
			THEN
				eStateEcGetSlaveNameSeq := eEcGetSlaveName_Start;
			END_IF

		eEcGetSlaveName_ErrorStep			:	(* Error detected *)

			bBusy := FALSE;
			bError := TRUE;

			IF NOT bExecute
			THEN
				fbEcGetAllSlaveAddr(bExecute 	:= FALSE);
				fbEcCoeSdoRead(		bExecute 	:= FALSE);
				
				bError 							:= FALSE;
				nErrId 							:= 0;
				
				eStateEcGetSlaveNameSeq 		:= eEcGetSlaveName_Start;
				eEcGetSlaveNameErrStep			:= eEcGetSlaveName_NoError;
			END_IF
		
	ELSE

		eStateEcGetSlaveNameSeq := eEcGetSlaveName_Start;
		eEcGetSlaveNameErrStep	:= eEcGetSlaveName_NoError;
	
	END_CASE

(* End *)

END_FUNCTION_BLOCK

// ---- POUs/TwinSAFE/Components/FB_TwinSafeConnectionEL2904.TcPOU
FUNCTION_BLOCK FB_TwinSafeConnectionEL2904
(*******************************************************************************************************
Description			:	Evaluate a TwinSAFE connection status and diagnosis to an EtherCAT terminal
Supported terminals : 	EL2904
Documentation 		:	EL2904 TwinSAFE output terminal with 4 fail-safe outputs
Version/Date 		:	V1.6.2/02.10.2015
Required libraries 	: 	TcSystem.lib (Tc2_System), TcEtherCAT.lib (Tc2_EtherCAT)
********************************************************************************************************)
VAR_INPUT
	
	tCoEReadCycle							:TIME 		:= T#0MS;			(* Read cycle CoE-Data, e.g. temperature *)

END_VAR
VAR_OUTPUT

	stInfoData						AT %I*	:ST_TsConnectionInfo1Byte;		(* EL6900 \ Connection Info Data \ Message_X Info Data*)
	nEcSlaveState					AT %I*	:UINT ;							(* EL2904 \ InfoData \ State *)
	stEcAdsAddr						AT %I*	:ST_AdsAddr;					(* EL2904 \ InfoData \ AdsAddr *)

(* act_EcSlaveIdentify *)
	sEcSlaveType							:STRING(15);
	sEcSlaveName							:STRING(31) := '';
	bSlaveIdentify							:BOOL;
	bSlaveTypeError							:BOOL;
	
(* act_Signals *)
	bChannel1								:BOOL;							
	bChannel2								:BOOL;
	bChannel3								:BOOL;
	bChannel4								:BOOL;

(* act_ConnectionState *)
	sState									:STRING;
	
(* act_ConnectionDiag *)
	sDiag									:STRING;
	sFault									:STRING(255);					(* FailSafe Error (Hardware)*)
	bError									:BOOL;							(* TwinSAFE-Error *)
	
(* act_ReadDiagObjects *)
	stSlaveTemp								:ST_TsSlave3Temp;
	bTempWarning							:BOOL;							(* Temperature warning: T1, T2, TOut*)
	stTsDiagObjectsBitsEL2904				:ST_TsDiagObjectsBitsEL2904;

END_VAR
VAR

(* act_ConnectionDiag *)
	nDiag0_3								:BYTE;

(* act_ReadDiagObjects *)
	eReadDiagObjState						:E_TsCycleDiagObj;
	eReadDiagObjErrStep						:E_TsCycleDiagObj := E_TsCycleDiagObj.eCycleDiagObj_NoError;
	bReadDiagObjError						:BOOL;							(* Error in the diagnosis objects read cycle *)  
	bReadDiagObjReset						:BOOL;							(* Reset the diagnosis objects read cycle error *)
	fbTimer									:TON;
	fbEcCoeSdoRead							:FB_EcCoESdoReadEx;
	stDiagObjects							:ST_TsDiagObjectsEL2904;

(* act_EcSlaveIdentify *)
	fbEcGetSlaveName						:FB_EcGetSlaveName;

END_VAR
VAR CONSTANT

(* act_ReadDiagObjects *)
	nWarningLevelTemp1						:INT	:= 85;					(* Temperature 1 warning level [°C] *)
	nWarningLevelTemp2						:INT	:= 85;					(* Temperature 2 warning level [°C] *)
	nWarningLevelTempOutputs				:INT	:= 85;					(* Temperature outputs warning level [°C] *)

END_VAR
(* End *)

(* Function Block TwinSAFE connection status and diagnosis for EL2904 Terminals *)

(* THIS CODE IS ONLY AN EXAMPLE - YOU HAVE TO CHECK APTITUDE FOR YOUR APPLICATION *)

	(* Identify the EtherCAT slave *)
		act_EcSlaveIdentify();

	(* Evaluate the connection state *)
		act_ConnectionState();
	
	(* Evaluate the connection diagnosis *)
		act_ConnectionDiag();
	
	(* Evaluate the EL2904 output signals *)
		act_Signals();
	
	(* Evaluate the Terminal temperatures and diagnostic objects *)
		IF bSlaveIdentify
		THEN
			act_ReadDiagObjects();
		ELSE
			eReadDiagObjState := E_TsCycleDiagObj.eCycleDiagObj_Init;
		END_IF
		
(* End *)

ACTION act_ConnectionDiag:
(* Evaluate the connection diagnosis *)

	(* Evaluate Bit 0..3 *)
	nDiag0_3 := USINT_TO_BYTE(stInfoData.nDiag) AND 16#0F;

	CASE nDiag0_3 OF
		0:		sDiag := 'No error';
		1:		sDiag := 'Invalid command';
		2:		sDiag := 'Unknown command';
		3:		sDiag := 'Invalid connection ID';
		4:		sDiag := 'Invalid CRC';
		5:		sDiag := 'Watchdog time elapsed';
		6:		sDiag := 'Invalid FSOE address';
		7:		sDiag := 'Invalid data';
		8:		sDiag := 'Invalid communication parameter length';
		9:		sDiag := 'Invalid communication parameters';
		10:		sDiag := 'Invalid user parameter length';
		11:		sDiag := 'Invalid user parameter';
		12:		sDiag := 'FSoE master reset';
		13:		sDiag := 'Module err detected on slave, with option "Module error is ComError" activated';
		14:		sDiag := 'Module err detected on EL290x, with option "Error acknowledge active" activated';
		15:		sDiag := 'Slave not yet started, or unexpected error argument';
	END_CASE

	(* Evaluate Bit 4..7 *)
	sFault:='';

	IF stInfoData.nDiag.4 
	THEN
		sFault	:= 'FSoE slave error detected - '; 
	END_IF

	IF stInfoData.nDiag.5 
	THEN
		sFault	:= concat(sFault,'FSoE slave reports Failsafe Value active - ');
	END_IF

	IF stInfoData.nDiag.6 
	THEN
		sFault	:= concat(sFault,'StartUp - ');
	END_IF

	IF stInfoData.nDiag.7 
	THEN
		sFault	:= concat(sFault, 'FSoE master reports Failsafe Value active');
	END_IF
		
	(* Error *)
	bError := stInfoData.nDiag <> 0;

(* End *)
END_ACTION

ACTION act_ConnectionState:
(* Evaluate the connection state *)

	CASE stInfoData.nState OF
		100:	sState := 'Reset state';
		101:	sState := 'Session state';
		102:	sState := 'Connection state';
		103:	sState := 'Parameter state';
		104:	sState := 'Data state';
		105:	sState := 'Shutdown state';
	ELSE
		sState := 'unknown';
	END_CASE
	
(* End *)
END_ACTION

ACTION act_DiagObjectsBits:
(* act_TsDiagObjectsBits *)

	stTsDiagObjectsBitsEL2904.bEsOrCcErrOutput1 			 := stDiagObjects.nErrorOutputs.0;
	stTsDiagObjectsBitsEL2904.bEsOrCcErrOutput2 			 := stDiagObjects.nErrorOutputs.1;
	stTsDiagObjectsBitsEL2904.bEsOrCcErrOutput3 			 := stDiagObjects.nErrorOutputs.2;
	stTsDiagObjectsBitsEL2904.bEsOrCcErrOutput4 			 := stDiagObjects.nErrorOutputs.3;
	stTsDiagObjectsBitsEL2904.bOlOrCvErrOutput1 			 := stDiagObjects.nErrorOutputs.4;
	stTsDiagObjectsBitsEL2904.bOlOrCvErrOutput2 			 := stDiagObjects.nErrorOutputs.5;
	stTsDiagObjectsBitsEL2904.bOlOrCvErrOutput3 			 := stDiagObjects.nErrorOutputs.6;
	stTsDiagObjectsBitsEL2904.bOlOrCvErrOutput4     		 := stDiagObjects.nErrorOutputs.7;

	stTsDiagObjectsBitsEL2904.bFieldVoltageTooHigh 			 := stDiagObjects.nSupplyError.0;
	stTsDiagObjectsBitsEL2904.bFieldVoltageTooLow  			 := stDiagObjects.nSupplyError.1;
	
	stTsDiagObjectsBitsEL2904.nOvertemperatureC1 			 := stDiagObjects.nTemperatureError.0;
	stTsDiagObjectsBitsEL2904.nOvertemperatureC2 			 := stDiagObjects.nTemperatureError.1;
	stTsDiagObjectsBitsEL2904.nOvertemperatureOutputs 		 := stDiagObjects.nTemperatureError.2;
	stTsDiagObjectsBitsEL2904.nTemperatureTooLowC1 			 := stDiagObjects.nTemperatureError.3;
	stTsDiagObjectsBitsEL2904.nTemperatureTooLowC2  		 := stDiagObjects.nTemperatureError.4;
	stTsDiagObjectsBitsEL2904.nTemperatureTooLowOutputs 	 := stDiagObjects.nTemperatureError.5;
	stTsDiagObjectsBitsEL2904.nOvertemperatureDiffBoard 	 := stDiagObjects.nTemperatureError.6;
	stTsDiagObjectsBitsEL2904.nOvertemperatureDiffBetwBoards := stDiagObjects.nTemperatureError.7;

(* End *)
END_ACTION

ACTION act_EcSlaveIdentify:
(* Identify the EtherCAT slave *)

	IF NOT nEcSlaveState.3
	THEN
		bSlaveIdentify  := FALSE;
		bSlaveTypeError := FALSE;
		sEcSlaveType    := '';
	END_IF

	IF nEcSlaveState.3
		AND NOT bSlaveIdentify
		AND NOT bSlaveTypeError
 		AND F_CreateAmsNetId(stEcAdsAddr.netId) <> '0.0.0.0.0.0' 
		AND stEcAdsAddr.port <> 0
	THEN

		fbEcCoeSdoRead(
			sNetId			:= 	F_CreateAmsNetId(stEcAdsAddr.netId),
			nSlaveAddr		:= 	stEcAdsAddr.port,
			nSubIndex		:= 	0,
			nIndex			:= 	16#1008,
			pDstBuf			:= 	ADR(sEcSlaveType),
			cbBufLen		:= 	SIZEOF(sEcSlaveType),
			bExecute		:= 	TRUE,
			tTimeout		:= 	DEFAULT_ADS_TIMEOUT);
	

		fbEcGetSlaveName(
			bExecute		:=	TRUE, 
			sNetId			:=	F_CreateAmsNetId(stEcAdsAddr.netId), 
			nSlaveAddr		:=	stEcAdsAddr.port, 
			tTimeout		:=	DEFAULT_ADS_TIMEOUT, 
			bBusy			=>	, 
			sSlaveName		=>	sEcSlaveName, 
			bError			=>	, 
			nErrId			=>	);

		IF NOT fbEcCoeSdoRead.bBusy
			AND NOT fbEcCoeSdoRead.bError
			AND NOT fbEcGetSlaveName.bBusy
			AND NOT fbEcGetSlaveName.bError
		THEN
		
			fbEcCoeSdoRead(bExecute := FALSE); 
			fbEcGetSlaveName(bExecute := FALSE); 

			IF sEcSlaveType = 'EL2904' 
				AND fbEcGetSlaveName.sSlaveName <> ''
			THEN
				bSlaveIdentify := TRUE;
			ELSE
				bSlaveTypeError := TRUE;
			END_IF

		ELSIF NOT fbEcCoeSdoRead.bBusy
			AND fbEcCoeSdoRead.bError
		OR (NOT fbEcGetSlaveName.bBusy
			AND fbEcGetSlaveName.bError)
		THEN
		
			fbEcCoeSdoRead(bExecute := FALSE); 
			fbEcGetSlaveName(bExecute := FALSE); 

		END_IF

	END_IF
	
(* End *)
END_ACTION

ACTION act_ReadDiagObjects:
(* Evaluate the Terminal temperatures and diagnostic objects *)

	CASE eReadDiagObjState OF

		eCycleDiagObj_Init				:	(* Init *)	

			IF nEcSlaveState.3					(* Slave in OP *)
				AND tCoEReadCycle <> T#0MS 		(* tCoEReadCycle <> t#0ms -> Read diagnostic aktiv *)
			THEN
				bReadDiagObjError := FALSE;
				fbEcCoeSdoRead(	bExecute := FALSE);
				fbTimer(IN := FALSE);
				eReadDiagObjState := eCycleDiagObj_ReadTemperature;
			END_IF

			
		eCycleDiagObj_ReadTemperature	:	(* Read temperature *)

			fbEcCoeSdoRead(
				sNetId			:= 	F_CreateAmsNetId(stEcAdsAddr.netId),
				nSlaveAddr		:= 	stEcAdsAddr.port,
				nSubIndex		:= 	1,
				nIndex			:= 	16#FA80,
				pDstBuf			:= 	ADR(stSlaveTemp),
				cbBufLen		:= 	SIZEOF(stSlaveTemp),
				bExecute		:= 	TRUE,
				tTimeout		:= 	DEFAULT_ADS_TIMEOUT,
				bCompleteAccess	:= 	TRUE);

			IF NOT fbEcCoeSdoRead.bBusy 
				AND NOT fbEcCoeSdoRead.bError 
			THEN
				fbEcCoeSdoRead(bExecute := FALSE);
				eReadDiagObjState := eCycleDiagObj_ReadDiag;
			ELSIF NOT fbEcCoeSdoRead.bBusy 
				AND fbEcCoeSdoRead.bError 
			THEN
				eReadDiagObjErrStep := eReadDiagObjState;
				eReadDiagObjState 	:= eCycleDiagObj_Error;
			END_IF

			
		eCycleDiagObj_ReadDiag			:	(* Read diacnostic objects *)

			fbTimer(IN := TRUE, PT := tCoEReadCycle);

			fbEcCoeSdoRead(
				sNetId			:= 	F_CreateAmsNetId(stEcAdsAddr.netId),
				nSlaveAddr		:= 	stEcAdsAddr.port,
				nSubIndex		:= 	1,
				nIndex			:= 	16#800E,
				pDstBuf			:= 	ADR(stDiagObjects),
				cbBufLen		:= 	SIZEOF(stDiagObjects),
				bExecute		:= 	TRUE,
				tTimeout		:= 	DEFAULT_ADS_TIMEOUT,
				bCompleteAccess	:= 	TRUE);

			IF NOT fbEcCoeSdoRead.bBusy 
				AND NOT fbEcCoeSdoRead.bError 
			THEN
				fbEcCoeSdoRead(bExecute := FALSE);
				act_DiagObjectsBits();
				eReadDiagObjState := eCycleDiagObj_ReadDelay;
			ELSIF NOT fbEcCoeSdoRead.bBusy 
				AND fbEcCoeSdoRead.bError 
			THEN
				eReadDiagObjErrStep := eReadDiagObjState;
				eReadDiagObjState 	:= eCycleDiagObj_Error;
			END_IF
				
			
		eCycleDiagObj_ReadDelay			:	(* Read delay *)
			fbTimer(
				IN := TRUE, 
				PT := tCoEReadCycle);

			IF fbTimer.Q 
			THEN
				fbTimer(IN := FALSE); 			
				eReadDiagObjState := eCycleDiagObj_Done;
			END_IF

			
		eCycleDiagObj_Done				:	(* Done *)

			eReadDiagObjState := eCycleDiagObj_Init;

			
		eCycleDiagObj_Error			:	(* Error detected *)

			bReadDiagObjError := TRUE;
		
			IF bReadDiagObjReset
			THEN
				bReadDiagObjError := FALSE;
				fbEcCoeSdoRead(bExecute := FALSE);
				eReadDiagObjErrStep := E_TsCycleDiagObj.eCycleDiagObj_NoError;
				eReadDiagObjState := eCycleDiagObj_Init;
			END_IF

	ELSE
		
		eReadDiagObjState := eCycleDiagObj_Init;
		
	END_CASE

	bTempWarning := stSlaveTemp.nInternalTemperature1 >= nWarningLevelTemp1 
						OR stSlaveTemp.nInternalTemperature2 >= nWarningLevelTemp2
							OR stSlaveTemp.nInternalTemperatureOutputs >= nWarningLevelTempOutputs;

(* End *)
END_ACTION

ACTION act_Signals:
(* Evaluate the output (EL2904) signals *)

	IF nEcSlaveState.3 (* Slave in operational state *)
	THEN
		(* OP -> transfer the signal states *)
		bChannel1 := stInfoData.nInOutSafeDataByte1.0;
		bChannel2 := stInfoData.nInOutSafeDataByte1.1;
		bChannel3 := stInfoData.nInOutSafeDataByte1.2;
		bChannel4 := stInfoData.nInOutSafeDataByte1.3;
	ELSE
		(* Error -> clear the signal states *)
		bChannel1 := bChannel2 := bChannel3 := bChannel4 := FALSE;
	END_IF

(* End *)
END_ACTION

END_FUNCTION_BLOCK

// ---- POUs/TwinSAFE/Components/FB_TwinSafeConnectionAX5805.TcPOU
FUNCTION_BLOCK FB_TwinSafeConnectionAX5805
(*******************************************************************************************************
Description			:	Evaluate a TwinSAFE connection status and diagnosis to an EtherCAT terminal
Supported terminals : 	AX5805(2 Axis)
Documentation 		:	AX5805 / AX5806 TwinSAFE drive option cards for the AX5000 servo drive
Version/Date 		:	V1.6.1/15.03.2016
Required libraries 	: 	TcSystem.lib (Tc2_System), TcEtherCAT.lib (Tc2_EtherCAT)
********************************************************************************************************)
VAR_INPUT
	
	tCoEReadCycle							:TIME 		:= T#0MS;			(* Read cycle CoE-Data, e.g. temperature *)

END_VAR
VAR_OUTPUT

	stInfoData						AT %I*	:ST_TsConnectionInfo8Byte;		(* EL6900 \ Connection Info Data \ Message_X Info Data*)
	nEcSlaveState					AT %I*	:UINT ;							(* AX5805 \ InfoData \ State *)
	stEcAdsAddr						AT %I*	:ST_AdsAddr;					(* AX5805 \ InfoData \ AdsAddr *)
	
(* act_EcSlaveIdentify *)
	sEcSlaveType							:STRING(15);
	sEcSlaveName							:STRING(31) := '';

	bSlaveIdentify							:BOOL;
	bSlaveTypeError							:BOOL;
	
(* act_Signals *)
	stSignalStatusMC1						:ST_TsStatusWordAX5805;
	stSignalControlStatusMC1				:ST_TsControlWordAX5805;
	stSignalStatusMC2						:ST_TsStatusWordAX5805;
	stSignalControlStatusMC2				:ST_TsControlWordAX5805;

(* act_ConnectionState *)
	sState									:STRING;
	
(* act_ConnectionDiag *)
	sDiag									:STRING;
	sFault									:STRING;						(* FailSafe Error (Hardware)*)
	bError									:BOOL;							(* TwinSAFE-Error *)
	
(* act_ReadDiagObjects *)
	stSlaveTemp								:ST_TsSlave2Temp;
	bTempWarning							:BOOL;							(* Temperature warning: T1, T2 *)

	eErrIndicesFA82ErrorMC1					:E_TsErrIndicesFA82AX5805;
	eErrIndicesFA82ErrorMC2					:E_TsErrIndicesFA82AX5805;
	eErrIndicesFA82DiagnosisMC1				:E_TsErrIndicesFA82AX5805;
	bErrIndicesFA82DiagnosisMC1Err			:BOOL;
	eErrIndicesFA82DiagnosisMC2				:E_TsErrIndicesFA82AX5805;
	bErrIndicesFA82DiagnosisMC2Err			:BOOL;	

	eDiagObjFA10LowByteMC1					:E_TsDiagnosisObjektsFA10AX5805;
	eDiagObjFA10HighByteMC1					:E_TsDiagnosisObjektsFA10AX5805;
	eDiagObjFA10LowByteMC2					:E_TsDiagnosisObjektsFA10AX5805;
	eDiagObjFA10HighByteMC2					:E_TsDiagnosisObjektsFA10AX5805;

END_VAR
VAR

(* act_ConnectionDiag *)
	nDiag0_3								:BYTE;

(* act_ReadDiagObjects *)
	eReadDiagObjState						:E_TsCycleDiagObj;
	eReadDiagObjErrStep						:E_TsCycleDiagObj := E_TsCycleDiagObj.eCycleDiagObj_NoError;
	bReadDiagObjError						:BOOL;								(* Error in the diagnosis objects read cycle *)  
	bReadDiagObjReset						:BOOL;								(* Reset the diagnosis objects read cycle error *)
	fbTimer									:TON;
	fbEcCoeSdoRead							:FB_EcCoESdoReadEx;
	stErrIndicesFA82						:ST_TsErrIndicesFA82AX5805;
	stDiagObjectsFA10						:ST_TsDiagObjectsFA10AX5805;

(* act_EcSlaveIdentify *)
	fbEcGetSlaveName						:FB_EcGetSlaveName;

END_VAR
VAR CONSTANT

(* act_ReadDiagObjects *)
	nWarningLevelTemp1						:INT	:= 85;						(* Temperature 1 warning level [°C] *)
	nWarningLevelTemp2						:INT	:= 85;						(* Temperature 2 warning level [°C] *)

END_VAR
(* End *)

(* Function Block TwinSAFE connection status and diagnosis for AX5805 Terminals *)

(* THIS CODE IS ONLY AN EXAMPLE - YOU HAVE TO CHECK APTITUDE FOR YOUR APPLICATION *)

	(* Identify the EtherCAT slave *)
		act_EcSlaveIdentify();

	(* Evaluate the connection state *)
		act_ConnectionState();
	
	(* Evaluate the connection diagnosis *)
		act_ConnectionDiag();
	
	(* Evaluate the AX5805 input and output signals *)
		act_Signals();
	
	(* Evaluate the Terminal temperatures and diagnostic objects *)
		IF bSlaveIdentify
		THEN
			act_ReadDiagObjects();
		ELSE
			eReadDiagObjState := E_TsCycleDiagObj.eCycleDiagObj_Init;
		END_IF
		
(* End *)

ACTION act_ConnectionDiag:
(* Evaluate the connection diagnosis *)

	(* Evaluate Bit 0..3 *)
	nDiag0_3 := USINT_TO_BYTE(stInfoData.nDiag) AND 16#0F;

	CASE nDiag0_3 OF
		0:		sDiag := 'No error';
		1:		sDiag := 'Invalid command';
		2:		sDiag := 'Unknown command';
		3:		sDiag := 'Invalid connection ID';
		4:		sDiag := 'Invalid CRC';
		5:		sDiag := 'Watchdog time elapsed';
		6:		sDiag := 'Invalid FSOE address';
		7:		sDiag := 'Invalid data';
		8:		sDiag := 'Invalid communication parameter length';
		9:		sDiag := 'Invalid communication parameters';
		10:		sDiag := 'Invalid user parameter length';
		11:		sDiag := 'Invalid user parameter';
		12:		sDiag := 'FSoE master reset';
		13:		sDiag := 'Module err detected on slave, with option "Module error is ComError" activated';
		14:		sDiag := 'Module err detected on EL290x, with option "Error acknowledge active" activated';
		15:		sDiag := 'Slave not yet started, or unexpected error argument';
	END_CASE

	(* Evaluate Bit 4..7 *)
	sFault:='';

	IF stInfoData.nDiag.4 
	THEN
		sFault	:= 'FSoE slave error detected - '; 
	END_IF

	IF stInfoData.nDiag.5 
	THEN
		sFault	:= concat(sFault,'FSoE slave reports Failsafe Value active - ');
	END_IF

	IF stInfoData.nDiag.6 
	THEN
		sFault	:= concat(sFault,'StartUp - ');
	END_IF

	IF stInfoData.nDiag.7 
	THEN
		sFault	:= concat(sFault, 'FSoE master reports Failsafe Value active');
	END_IF
		
	(* Error *)
	bError := stInfoData.nDiag <> 0;

(* End *)
END_ACTION

ACTION act_ConnectionState:
(* Evaluate the connection state *)

	CASE stInfoData.nState OF
		100:	sState := 'Reset state';
		101:	sState := 'Session state';
		102:	sState := 'Connection state';
		103:	sState := 'Parameter state';
		104:	sState := 'Data state';
		105:	sState := 'Shutdown state';
	ELSE
		sState := 'unknown';
	END_CASE
	
(* End *)
END_ACTION

ACTION act_EcSlaveIdentify:
(* Identify the EtherCAT slave *)

	IF NOT nEcSlaveState.3
	THEN
		bSlaveIdentify  := FALSE;
		bSlaveTypeError := FALSE;
		sEcSlaveType    := '';
	END_IF

	IF nEcSlaveState.3
		AND NOT bSlaveIdentify
		AND NOT bSlaveTypeError
		AND F_CreateAmsNetId(stEcAdsAddr.netId) <> '0.0.0.0.0.0' 
		AND stEcAdsAddr.port <> 0
	THEN

		fbEcCoeSdoRead(
			sNetId			:= 	F_CreateAmsNetId(stEcAdsAddr.netId),
			nSlaveAddr		:= 	stEcAdsAddr.port,
			nSubIndex		:= 	0,
			nIndex			:= 	16#1008,
			pDstBuf			:= 	ADR(sEcSlaveType),
			cbBufLen		:= 	SIZEOF(sEcSlaveType),
			bExecute		:= 	TRUE,
			tTimeout		:= 	DEFAULT_ADS_TIMEOUT);
	

		fbEcGetSlaveName(
			bExecute		:=	TRUE, 
			sNetId			:=	F_CreateAmsNetId(stEcAdsAddr.netId), 
			nSlaveAddr		:=	stEcAdsAddr.port, 
			tTimeout		:=	DEFAULT_ADS_TIMEOUT, 
			bBusy			=>	, 
			sSlaveName		=>	sEcSlaveName, 
			bError			=>	, 
			nErrId			=>	);

		IF NOT fbEcCoeSdoRead.bBusy
			AND NOT fbEcCoeSdoRead.bError
			AND NOT fbEcGetSlaveName.bBusy
			AND NOT fbEcGetSlaveName.bError
		THEN
		
			fbEcCoeSdoRead(bExecute := FALSE); 
			fbEcGetSlaveName(bExecute := FALSE); 

			IF sEcSlaveType = 'AX5805' 
				AND fbEcGetSlaveName.sSlaveName <> ''
			THEN
				bSlaveIdentify := TRUE;
			ELSE
				bSlaveTypeError := TRUE;
			END_IF

		ELSIF NOT fbEcCoeSdoRead.bBusy
			AND fbEcCoeSdoRead.bError
		OR (NOT fbEcGetSlaveName.bBusy
			AND fbEcGetSlaveName.bError)
		THEN
		
			fbEcCoeSdoRead(bExecute := FALSE); 
			fbEcGetSlaveName(bExecute := FALSE); 

		END_IF

	END_IF
	
(* End *)
END_ACTION

ACTION act_ReadDiagObjects:
(* Evaluate the Terminal temperatures and diagnostic objects *)

	CASE eReadDiagObjState OF

		eCycleDiagObj_Init				:	(* Init *)	

			IF nEcSlaveState.3					(* Slave in OP *)
				AND tCoEReadCycle <> T#0MS 		(* tCoEReadCycle <> t#0ms -> Read diagnostic aktiv *)
			THEN
				bReadDiagObjError := FALSE;
				fbEcCoeSdoRead(	bExecute := FALSE);
				fbTimer(IN := FALSE);
				eReadDiagObjState := eCycleDiagObj_ReadTemperature;
			END_IF

			
		eCycleDiagObj_ReadTemperature	:	(* Read temperature *)

			fbEcCoeSdoRead(
				sNetId			:= 	F_CreateAmsNetId(stEcAdsAddr.netId),
				nSlaveAddr		:= 	stEcAdsAddr.port,
				nSubIndex		:= 	1,
				nIndex			:= 	16#FA80,
				pDstBuf			:= 	ADR(stSlaveTemp),
				cbBufLen		:= 	SIZEOF(stSlaveTemp),
				bExecute		:= 	TRUE,
				tTimeout		:= 	DEFAULT_ADS_TIMEOUT,
				bCompleteAccess	:= 	TRUE);

			IF NOT fbEcCoeSdoRead.bBusy 
				AND NOT fbEcCoeSdoRead.bError 
			THEN
				fbEcCoeSdoRead(bExecute := FALSE);
				eReadDiagObjState := eCycleDiagObj_ReadErrorIndices;
			ELSIF NOT fbEcCoeSdoRead.bBusy 
				AND fbEcCoeSdoRead.bError 
			THEN
				eReadDiagObjErrStep := eReadDiagObjState;
				eReadDiagObjState 	:= eCycleDiagObj_Error;
			END_IF

			
		eCycleDiagObj_ReadErrorIndices			:	(* Read error indices *)

			fbTimer(IN := TRUE, PT := tCoEReadCycle);

			fbEcCoeSdoRead(
				sNetId			:= 	F_CreateAmsNetId(stEcAdsAddr.netId),
				nSlaveAddr		:= 	stEcAdsAddr.port,
				nSubIndex		:= 	1,
				nIndex			:= 	16#FA82,
				pDstBuf			:= 	ADR(stErrIndicesFA82),
				cbBufLen		:= 	SIZEOF(stErrIndicesFA82),
				bExecute		:= 	TRUE,
				tTimeout		:= 	DEFAULT_ADS_TIMEOUT,
				bCompleteAccess	:= 	TRUE);

			IF NOT fbEcCoeSdoRead.bBusy 
				AND NOT fbEcCoeSdoRead.bError 
			THEN
				fbEcCoeSdoRead(bExecute := FALSE);

				eErrIndicesFA82ErrorMC1 	 	:= stErrIndicesFA82.nErrorMC1;
				eErrIndicesFA82ErrorMC2 	 	:= stErrIndicesFA82.nErrorMC2;
				eErrIndicesFA82DiagnosisMC1 	:= stErrIndicesFA82.nDiagnosisMC1;
				bErrIndicesFA82DiagnosisMC1Err 	:= eErrIndicesFA82DiagnosisMC1 <> E_TsErrIndicesFA82AX5805.eAX5805FA82_NoError;
				eErrIndicesFA82DiagnosisMC2 	:= stErrIndicesFA82.nDiagnosisMC2;
				bErrIndicesFA82DiagnosisMC2Err 	:= eErrIndicesFA82DiagnosisMC2 <> E_TsErrIndicesFA82AX5805.eAX5805FA82_NoError;
				
				eReadDiagObjState := eCycleDiagObj_ReadDiag;
			ELSIF NOT fbEcCoeSdoRead.bBusy 
				AND fbEcCoeSdoRead.bError 
			THEN
				eReadDiagObjErrStep := eReadDiagObjState;
				eReadDiagObjState 	:= eCycleDiagObj_Error;
			END_IF
				
			
		eCycleDiagObj_ReadDiag			:	(* Read diacnostic objects *)

			fbTimer(IN := TRUE, PT := tCoEReadCycle);

			fbEcCoeSdoRead(
				sNetId			:= 	F_CreateAmsNetId(stEcAdsAddr.netId),
				nSlaveAddr		:= 	stEcAdsAddr.port,
				nSubIndex		:= 	1,
				nIndex			:= 	16#FA10,
				pDstBuf			:= 	ADR(stDiagObjectsFA10),
				cbBufLen		:= 	SIZEOF(stDiagObjectsFA10),
				bExecute		:= 	TRUE,
				tTimeout		:= 	DEFAULT_ADS_TIMEOUT,
				bCompleteAccess	:= 	TRUE);

			IF NOT fbEcCoeSdoRead.bBusy 
				AND NOT fbEcCoeSdoRead.bError 
			THEN
				fbEcCoeSdoRead(bExecute := FALSE);
				
				eDiagObjFA10LowByteMC1	:=	TO_WORD(stDiagObjectsFA10.nReasonForShutdownAxis1) AND 16#00FF;	
				eDiagObjFA10HighByteMC1	:=	TO_WORD(stDiagObjectsFA10.nReasonForShutdownAxis1) AND 16#FF00;	
				eDiagObjFA10LowByteMC2	:=	TO_WORD(stDiagObjectsFA10.nReasonForShutdownAxis2) AND 16#00FF;	
				eDiagObjFA10HighByteMC2	:=	TO_WORD(stDiagObjectsFA10.nReasonForShutdownAxis2) AND 16#FF00;	
				
				eReadDiagObjState := eCycleDiagObj_ReadDelay;
			ELSIF NOT fbEcCoeSdoRead.bBusy 
				AND fbEcCoeSdoRead.bError 
			THEN
				eReadDiagObjErrStep := eReadDiagObjState;
				eReadDiagObjState 	:= eCycleDiagObj_Error;
			END_IF
				
			
		eCycleDiagObj_ReadDelay		:	(* Read delay *)
			fbTimer(
				IN := TRUE, 
				PT := tCoEReadCycle);

